LIN {X 0,Y 448.323,Z 386.523,A -85,B 0,C 180,E1 21192.232,E2 21192.232} C_VEL
LIN {X 0,Y 450.072,Z 390.704,A -85,B 0,C 180,E1 21190.556,E2 21190.556} C_VEL
LIN {X 0,Y 452.534,Z 396.687,A -85,B 0,C 180,E1 21188.745,E2 21188.745} C_VEL
LIN {X 0,Y 455.532,Z 405.377,A -85,B 0,C 180,E1 21186.76,E2 21186.76} C_VEL
LIN {X 0,Y 458.055,Z 414.218,A -85,B 0,C 180,E1 21185.151,E2 21185.151} C_VEL
LIN {X 0,Y 453.671,Z 442.774,A -85,B 0,C 180,E1 21182.083,E2 21182.083} C_VEL
LIN {X 0,Y 451.675,Z 461.261,A -85,B 0,C 180,E1 21180.253,E2 21180.253} C_VEL
LIN {X 0,Y 454.574,Z 485.875,A -85,B 0,C 180,E1 21179.545,E2 21179.545} C_VEL
LIN {X 0,Y 450.23,Z 669.654,A -85,B 0,C 180,E1 21176.099,E2 21176.099} C_VEL
LIN {X 0,Y 449.356,Z 688.845,A -85,B 0,C 180,E1 21175.507,E2 21175.507} C_VEL
LIN {X 0,Y 448.327,Z 706.902,A -85,B 0,C 180,E1 21174.719,E2 21174.719} C_VEL
LIN {X 0,Y 447.086,Z 725.176,A -85,B 0,C 180,E1 21173.668,E2 21173.668} C_VEL
LIN {X 0,Y 445.807,Z 742.394,A -85,B 0,C 180,E1 21172.413,E2 21172.413} C_VEL
LIN {X 0,Y 444.541,Z 758.619,A -85,B 0,C 180,E1 21170.954,E2 21170.954} C_VEL
LIN {X 0,Y 443.391,Z 773.227,A -85,B 0,C 180,E1 21169.359,E2 21169.359} C_VEL
LIN {X 0,Y 442.317,Z 787.369,A -85,B 0,C 180,E1 21167.497,E2 21167.497} C_VEL
LIN {X 0,Y 441.437,Z 799.818,A -85,B 0,C 180,E1 21165.502,E2 21165.502} C_VEL
LIN {X 0,Y 440.821,Z 810.693,A -85,B 0,C 180,E1 21163.377,E2 21163.377} C_VEL
LIN {X 0,Y 440.407,Z 819.525,A -85,B 0,C 180,E1 21161.254,E2 21161.254} C_VEL
LIN {X 0,Y 440.196,Z 826.898,A -85,B 0,C 180,E1 21159.017,E2 21159.017} C_VEL
LIN {X 0,Y 440.132,Z 832.486,A -85,B 0,C 180,E1 21156.784,E2 21156.784} C_VEL
LIN {X 0,Y 440.129,Z 836.41,A -85,B 0,C 180,E1 21154.561,E2 21154.561} C_VEL
LIN {X 0,Y 440.162,Z 838.826,A -85,B 0,C 180,E1 21152.213,E2 21152.213} C_VEL
LIN {X 0,Y 440.188,Z 839.52,A -85,B 0,C 180,E1 21149.87,E2 21149.87} C_VEL
LIN {X 0,Y 440.167,Z 838.494,A -85,B 0,C 180,E1 21147.526,E2 21147.526} C_VEL
LIN {X 0,Y 440.145,Z 835.73,A -85,B 0,C 180,E1 21145.179,E2 21145.179} C_VEL
LIN {X 0,Y 440.157,Z 831.15,A -85,B 0,C 180,E1 21142.823,E2 21142.823} C_VEL
LIN {X 0,Y 440.234,Z 825.056,A -85,B 0,C 180,E1 21140.588,E2 21140.588} C_VEL
LIN {X 0,Y 440.458,Z 817.062,A -85,B 0,C 180,E1 21138.344,E2 21138.344} C_VEL
LIN {X 0,Y 440.871,Z 807.59,A -85,B 0,C 180,E1 21136.224,E2 21136.224} C_VEL
LIN {X 0,Y 441.467,Z 796.714,A -85,B 0,C 180,E1 21134.23,E2 21134.23} C_VEL
LIN {X 0,Y 442.299,Z 783.981,A -85,B 0,C 180,E1 21132.299,E2 21132.299} C_VEL
LIN {X 0,Y 443.301,Z 769.666,A -85,B 0,C 180,E1 21130.5,E2 21130.5} C_VEL
LIN {X 0,Y 444.48,Z 753.65,A -85,B 0,C 180,E1 21128.835,E2 21128.835} C_VEL
LIN {X 0,Y 445.682,Z 737.336,A -85,B 0,C 180,E1 21127.441,E2 21127.441} C_VEL
LIN {X 0,Y 446.939,Z 719.499,A -85,B 0,C 180,E1 21126.203,E2 21126.203} C_VEL
LIN {X 0,Y 448.18,Z 700.55,A -85,B 0,C 180,E1 21125.167,E2 21125.167} C_VEL
LIN {X 0,Y 449.289,Z 680.808,A -85,B 0,C 180,E1 21124.364,E2 21124.364} C_VEL
LIN {X 0,Y 450.185,Z 660.789,A -85,B 0,C 180,E1 21123.804,E2 21123.804} C_VEL
LIN {X 0,Y 453.255,Z 560.014,A -85,B 0,C 180,E1 21121.719,E2 21121.719} C_VEL
LIN {X 0,Y 456.39,Z 483.809,A -85,B 0,C 180,E1 21119.981,E2 21119.981} C_VEL
LIN {X 0,Y 453.832,Z 456.502,A -85,B 0,C 180,E1 21118.93,E2 21118.93} C_VEL
LIN {X 0,Y 452.06,Z 438.943,A -85,B 0,C 180,E1 21118.138,E2 21118.138} C_VEL
LIN {X 0,Y 454.372,Z 409.393,A -85,B 0,C 180,E1 21115.386,E2 21115.386} C_VEL
LIN {X 0,Y 446.459,Z 386.782,A -85,B 0,C 180,E1 21112.447,E2 21112.447} C_VEL
LIN {X 0,Y 441.13,Z 371.851,A -85,B 0,C 180,E1 21110.354,E2 21110.354} C_VEL
LIN {X 0,Y 441.125,Z 371.85,A -85,B 0,C 180,E1 21106.624,E2 21106.624} C_VEL
LIN {X 0,Y 441.137,Z 371.849,A -85,B 0,C 180,E1 21102.937,E2 21102.937} C_VEL
LIN {X 0,Y 441.181,Z 371.846,A -85,B 0,C 180,E1 21099.388,E2 21099.388} C_VEL
LIN {X 0,Y 441.156,Z 372.028,A -85,B 0,C 180,E1 21098.847,E2 21098.847} C_VEL
LIN {X 0,Y 442.405,Z 375.286,A -85,B 0,C 180,E1 21098.097,E2 21098.097} C_VEL
LIN {X 0,Y 444.147,Z 377.5,A -85,B 0,C 180,E1 21097.432,E2 21097.432} C_VEL
LIN {X 0,Y 445.923,Z 381.17,A -85,B 0,C 180,E1 21096.609,E2 21096.609} C_VEL
LIN {X 0,Y 448.955,Z 387.643,A -85,B 0,C 180,E1 21095.291,E2 21095.291} C_VEL
LIN {X 0,Y 452.423,Z 396,A -85,B 0,C 180,E1 21093.802,E2 21093.802} C_VEL
LIN {X 0,Y 455.852,Z 406.812,A -85,B 0,C 180,E1 21092.151,E2 21092.151} C_VEL
LIN {X 0,Y 456.831,Z 411.358,A -85,B 0,C 180,E1 21091.54,E2 21091.54} C_VEL
LIN {X 0,Y 456.708,Z 416.112,A -85,B 0,C 180,E1 21091.109,E2 21091.109} C_VEL
LIN {X 0,Y 459.041,Z 430.919,A -85,B 0,C 180,E1 21090.399,E2 21090.399} C_VEL
LIN {X 0,Y 454.36,Z 526.982,A -85,B 0,C 180,E1 21088.206,E2 21088.206} C_VEL
LIN {X 0,Y 451.215,Z 624.113,A -85,B 0,C 180,E1 21086.148,E2 21086.148} C_VEL
LIN {X 0,Y 450.426,Z 643.02,A -85,B 0,C 180,E1 21085.508,E2 21085.508} C_VEL
LIN {X 0,Y 449.445,Z 661.366,A -85,B 0,C 180,E1 21084.653,E2 21084.653} C_VEL
LIN {X 0,Y 448.235,Z 679.768,A -85,B 0,C 180,E1 21083.534,E2 21083.534} C_VEL
LIN {X 0,Y 447.001,Z 696.185,A -85,B 0,C 180,E1 21082.28,E2 21082.28} C_VEL
LIN {X 0,Y 445.732,Z 711.737,A -85,B 0,C 180,E1 21080.827,E2 21080.827} C_VEL
LIN {X 0,Y 444.47,Z 726.31,A -85,B 0,C 180,E1 21079.174,E2 21079.174} C_VEL
LIN {X 0,Y 443.285,Z 739.778,A -85,B 0,C 180,E1 21077.321,E2 21077.321} C_VEL
LIN {X 0,Y 442.267,Z 751.622,A -85,B 0,C 180,E1 21075.338,E2 21075.338} C_VEL
LIN {X 0,Y 441.446,Z 761.933,A -85,B 0,C 180,E1 21073.224,E2 21073.224} C_VEL
LIN {X 0,Y 440.859,Z 770.262,A -85,B 0,C 180,E1 21071.115,E2 21071.115} C_VEL
LIN {X 0,Y 440.452,Z 777.21,A -85,B 0,C 180,E1 21068.88,E2 21068.88} C_VEL
LIN {X 0,Y 440.201,Z 782.678,A -85,B 0,C 180,E1 21066.521,E2 21066.521} C_VEL
LIN {X 0,Y 440.076,Z 786.425,A -85,B 0,C 180,E1 21064.115,E2 21064.115} C_VEL
LIN {X 0,Y 440.031,Z 788.434,A -85,B 0,C 180,E1 21061.693,E2 21061.693} C_VEL
LIN {X 0,Y 440.027,Z 788.727,A -85,B 0,C 180,E1 21059.349,E2 21059.349} C_VEL
LIN {X 0,Y 440.037,Z 787.283,A -85,B 0,C 180,E1 21056.874,E2 21056.874} C_VEL
LIN {X 0,Y 440.1,Z 784.224,A -85,B 0,C 180,E1 21054.524,E2 21054.524} C_VEL
LIN {X 0,Y 440.26,Z 779.442,A -85,B 0,C 180,E1 21052.168,E2 21052.168} C_VEL
LIN {X 0,Y 440.55,Z 773.222,A -85,B 0,C 180,E1 21049.935,E2 21049.935} C_VEL
LIN {X 0,Y 441.035,Z 765.18,A -85,B 0,C 180,E1 21047.695,E2 21047.695} C_VEL
LIN {X 0,Y 441.71,Z 755.698,A -85,B 0,C 180,E1 21045.582,E2 21045.582} C_VEL
LIN {X 0,Y 442.573,Z 744.828,A -85,B 0,C 180,E1 21043.596,E2 21043.596} C_VEL
LIN {X 0,Y 443.616,Z 732.581,A -85,B 0,C 180,E1 21041.742,E2 21041.742} C_VEL
LIN {X 0,Y 444.834,Z 718.548,A -85,B 0,C 180,E1 21039.976,E2 21039.976} C_VEL
LIN {X 0,Y 446.148,Z 703.004,A -85,B 0,C 180,E1 21038.367,E2 21038.367} C_VEL
LIN {X 0,Y 447.44,Z 686.629,A -85,B 0,C 180,E1 21036.979,E2 21036.979} C_VEL
LIN {X 0,Y 448.687,Z 669.284,A -85,B 0,C 180,E1 21035.793,E2 21035.793} C_VEL
LIN {X 0,Y 449.812,Z 650.874,A -85,B 0,C 180,E1 21034.806,E2 21034.806} C_VEL
LIN {X 0,Y 450.73,Z 631.633,A -85,B 0,C 180,E1 21034.038,E2 21034.038} C_VEL
LIN {X 0,Y 451.401,Z 612.37,A -85,B 0,C 180,E1 21033.516,E2 21033.516} C_VEL
LIN {X 0,Y 455.727,Z 428.996,A -85,B 0,C 180,E1 21030.112,E2 21030.112} C_VEL
LIN {X 0,Y 452.048,Z 408.245,A -85,B 0,C 180,E1 21029.421,E2 21029.421} C_VEL
LIN {X 0,Y 452.04,Z 405.292,A -85,B 0,C 180,E1 21029.117,E2 21029.117} C_VEL
LIN {X 0,Y 445.696,Z 385.318,A -85,B 0,C 180,E1 21026.568,E2 21026.568} C_VEL
LIN {X 0,Y 441.168,Z 371.843,A -85,B 0,C 180,E1 21024.774,E2 21024.774} C_VEL
LIN {X 0,Y 441.138,Z 371.849,A -85,B 0,C 180,E1 21021.109,E2 21021.109} C_VEL
LIN {X 0,Y 441.128,Z 371.847,A -85,B 0,C 180,E1 21017.447,E2 21017.447} C_VEL
LIN {X 0,Y 441.133,Z 371.847,A -85,B 0,C 180,E1 21013.694,E2 21013.694} C_VEL
LIN {X 0,Y 441.158,Z 371.846,A -85,B 0,C 180,E1 21010.066,E2 21010.066} C_VEL
LIN {X 0,Y 441.182,Z 371.844,A -85,B 0,C 180,E1 21008.299,E2 21008.299} C_VEL
LIN {X 0,Y 440.154,Z 371.972,A -85,B 0,C 180,E1 21007.299,E2 21007.299} C_VEL
LIN {X 0,Y 433.661,Z 372.783,A -85,B 0,C 180,E1 21004.411,E2 21004.411} C_VEL
LIN {X 0,Y 433.201,Z 372.837,A -85,B 0,C 180,E1 21003.749,E2 21003.749} C_VEL
LIN {X 0,Y 433.227,Z 372.834,A -85,B 0,C 180,E1 21000.055,E2 21000.055} C_VEL
LIN {X 0,Y 433.237,Z 372.832,A -85,B 0,C 180,E1 20996.303,E2 20996.303} C_VEL
LIN {X 0,Y 433.218,Z 372.833,A -85,B 0,C 180,E1 20992.527,E2 20992.527} C_VEL
LIN {X 0,Y 433.195,Z 372.835,A -85,B 0,C 180,E1 20988.853,E2 20988.853} C_VEL
LIN {X 0,Y 433.185,Z 372.836,A -85,B 0,C 180,E1 20985.119,E2 20985.119} C_VEL
LIN {X 0,Y 433.191,Z 372.835,A -85,B 0,C 180,E1 20981.314,E2 20981.314} C_VEL
LIN {X 0,Y 433.215,Z 372.834,A -85,B 0,C 180,E1 20977.693,E2 20977.693} C_VEL
LIN {X 0,Y 433.234,Z 372.83,A -85,B 0,C 180,E1 20973.97,E2 20973.97} C_VEL
LIN {X 0,Y 433.23,Z 372.834,A -85,B 0,C 180,E1 20970.132,E2 20970.132} C_VEL
LIN {X 0,Y 433.201,Z 372.831,A -85,B 0,C 180,E1 20966.427,E2 20966.427} C_VEL
LIN {X 0,Y 433.184,Z 372.831,A -85,B 0,C 180,E1 20962.84,E2 20962.84} C_VEL
LIN {X 0,Y 433.189,Z 372.834,A -85,B 0,C 180,E1 20959.09,E2 20959.09} C_VEL
LIN {X 0,Y 433.212,Z 372.836,A -85,B 0,C 180,E1 20955.429,E2 20955.429} C_VEL
LIN {X 0,Y 433.238,Z 372.836,A -85,B 0,C 180,E1 20951.707,E2 20951.707} C_VEL
LIN {X 0,Y 433.231,Z 372.833,A -85,B 0,C 180,E1 20947.902,E2 20947.902} C_VEL
LIN {X 0,Y 433.204,Z 372.834,A -85,B 0,C 180,E1 20944.137,E2 20944.137} C_VEL
LIN {X 0,Y 433.187,Z 372.834,A -85,B 0,C 180,E1 20940.479,E2 20940.479} C_VEL
LIN {X 0,Y 433.185,Z 372.838,A -85,B 0,C 180,E1 20936.674,E2 20936.674} C_VEL
LIN {X 0,Y 433.196,Z 372.839,A -85,B 0,C 180,E1 20932.957,E2 20932.957} C_VEL
LIN {X 0,Y 433.235,Z 372.836,A -85,B 0,C 180,E1 20929.396,E2 20929.396} C_VEL
LIN {X 0,Y 433.227,Z 372.835,A -85,B 0,C 180,E1 20925.628,E2 20925.628} C_VEL
LIN {X 0,Y 433.21,Z 372.837,A -85,B 0,C 180,E1 20921.838,E2 20921.838} C_VEL
LIN {X 0,Y 433.185,Z 372.838,A -85,B 0,C 180,E1 20918.213,E2 20918.213} C_VEL
LIN {X 0,Y 433.199,Z 372.944,A -85,B 0,C 180,E1 20914.514,E2 20914.514} C_VEL
LIN {X 0,Y 438.764,Z 393.227,A -85,B 0,C 180,E1 20911.037,E2 20911.037} C_VEL
LIN {X 0,Y 441.094,Z 402.817,A -85,B 0,C 180,E1 20909.465,E2 20909.465} C_VEL
LIN {X 0,Y 439.171,Z 430.368,A -85,B 0,C 180,E1 20905.631,E2 20905.631} C_VEL
LIN {X 0,Y 437.342,Z 459.208,A -85,B 0,C 180,E1 20901.672,E2 20901.672} C_VEL
LIN {X 0,Y 436.291,Z 479.402,A -85,B 0,C 180,E1 20898.979,E2 20898.979} C_VEL
LIN {X 0,Y 439.269,Z 500.885,A -85,B 0,C 180,E1 20898.376,E2 20898.376} C_VEL
LIN {X 0,Y 437.139,Z 601.136,A -85,B 0,C 180,E1 20896.315,E2 20896.315} C_VEL
LIN {X 0,Y 436.787,Z 616.364,A -85,B 0,C 180,E1 20895.773,E2 20895.773} C_VEL
LIN {X 0,Y 436.267,Z 632.271,A -85,B 0,C 180,E1 20894.942,E2 20894.942} C_VEL
LIN {X 0,Y 435.587,Z 647.652,A -85,B 0,C 180,E1 20893.839,E2 20893.839} C_VEL
LIN {X 0,Y 434.95,Z 661.323,A -85,B 0,C 180,E1 20892.547,E2 20892.547} C_VEL
LIN {X 0,Y 434.38,Z 672.936,A -85,B 0,C 180,E1 20891.149,E2 20891.149} C_VEL
LIN {X 0,Y 433.908,Z 682.701,A -85,B 0,C 180,E1 20889.684,E2 20889.684} C_VEL
LIN {X 0,Y 433.496,Z 691.731,A -85,B 0,C 180,E1 20887.955,E2 20887.955} C_VEL
LIN {X 0,Y 433.223,Z 698.656,A -85,B 0,C 180,E1 20886.228,E2 20886.228} C_VEL
LIN {X 0,Y 433.06,Z 704.17,A -85,B 0,C 180,E1 20884.37,E2 20884.37} C_VEL
LIN {X 0,Y 432.988,Z 708,A -85,B 0,C 180,E1 20882.382,E2 20882.382} C_VEL
LIN {X 0,Y 433.023,Z 709.862,A -85,B 0,C 180,E1 20880.529,E2 20880.529} C_VEL
LIN {X 0,Y 433.109,Z 710.028,A -85,B 0,C 180,E1 20878.545,E2 20878.545} C_VEL
LIN {X 0,Y 433.284,Z 708.445,A -85,B 0,C 180,E1 20876.693,E2 20876.693} C_VEL
LIN {X 0,Y 433.567,Z 704.888,A -85,B 0,C 180,E1 20874.707,E2 20874.707} C_VEL
LIN {X 0,Y 433.969,Z 699.603,A -85,B 0,C 180,E1 20872.853,E2 20872.853} C_VEL
LIN {X 0,Y 434.461,Z 692.85,A -85,B 0,C 180,E1 20871.13,E2 20871.13} C_VEL
LIN {X 0,Y 435.104,Z 683.912,A -85,B 0,C 180,E1 20869.407,E2 20869.407} C_VEL
LIN {X 0,Y 435.857,Z 673.21,A -85,B 0,C 180,E1 20867.816,E2 20867.816} C_VEL
LIN {X 0,Y 436.602,Z 662.003,A -85,B 0,C 180,E1 20866.492,E2 20866.492} C_VEL
LIN {X 0,Y 437.373,Z 649.291,A -85,B 0,C 180,E1 20865.3,E2 20865.3} C_VEL
LIN {X 0,Y 438.171,Z 634.655,A -85,B 0,C 180,E1 20864.244,E2 20864.244} C_VEL
LIN {X 0,Y 438.804,Z 620.091,A -85,B 0,C 180,E1 20863.452,E2 20863.452} C_VEL
LIN {X 0,Y 439.375,Z 603.875,A -85,B 0,C 180,E1 20862.822,E2 20862.822} C_VEL
LIN {X 0,Y 443.897,Z 510.297,A -85,B 0,C 180,E1 20860.295,E2 20860.295} C_VEL
LIN {X 0,Y 444.177,Z 501.591,A -85,B 0,C 180,E1 20860.039,E2 20860.039} C_VEL
LIN {X 0,Y 440.597,Z 481.46,A -85,B 0,C 180,E1 20859.048,E2 20859.048} C_VEL
LIN {X 0,Y 440.178,Z 478.915,A -85,B 0,C 180,E1 20858.888,E2 20858.888} C_VEL
LIN {X 0,Y 443.155,Z 451.096,A -85,B 0,C 180,E1 20854.759,E2 20854.759} C_VEL
LIN {X 0,Y 446.814,Z 425.609,A -85,B 0,C 180,E1 20850.777,E2 20850.777} C_VEL
LIN {X 0,Y 448.475,Z 415.609,A -85,B 0,C 180,E1 20849.132,E2 20849.132} C_VEL
LIN {X 0,Y 446.478,Z 406.377,A -85,B 0,C 180,E1 20846.878,E2 20846.878} C_VEL
LIN {X 0,Y 444.585,Z 399.623,A -85,B 0,C 180,E1 20844.849,E2 20844.849} C_VEL
LIN {X 0,Y 442.913,Z 394.174,A -85,B 0,C 180,E1 20842.771,E2 20842.771} C_VEL
LIN {X 0,Y 441.579,Z 390.597,A -85,B 0,C 180,E1 20840.822,E2 20840.822} C_VEL
LIN {X 0,Y 440.717,Z 387.966,A -85,B 0,C 180,E1 20838.28,E2 20838.28} C_VEL
LIN {X 0,Y 440.834,Z 387.574,A -85,B 0,C 180,E1 20836.347,E2 20836.347} C_VEL
LIN {X 0,Y 441.244,Z 389.399,A -85,B 0,C 180,E1 20834.261,E2 20834.261} C_VEL
LIN {X 0,Y 442.742,Z 392.108,A -85,B 0,C 180,E1 20832.398,E2 20832.398} C_VEL
LIN {X 0,Y 444.376,Z 396.253,A -85,B 0,C 180,E1 20830.689,E2 20830.689} C_VEL
LIN {X 0,Y 446.617,Z 401.89,A -85,B 0,C 180,E1 20828.926,E2 20828.926} C_VEL
LIN {X 0,Y 449.341,Z 410.137,A -85,B 0,C 180,E1 20826.981,E2 20826.981} C_VEL
LIN {X 0,Y 451.373,Z 417.564,A -85,B 0,C 180,E1 20825.555,E2 20825.555} C_VEL
LIN {X 0,Y 446.824,Z 444.559,A -85,B 0,C 180,E1 20822.559,E2 20822.559} C_VEL
LIN {X 0,Y 444.658,Z 462.787,A -85,B 0,C 180,E1 20820.706,E2 20820.706} C_VEL
LIN {X 0,Y 447.451,Z 486.897,A -85,B 0,C 180,E1 20819.997,E2 20819.997} C_VEL
LIN {X 0,Y 442.821,Z 669.243,A -85,B 0,C 180,E1 20816.493,E2 20816.493} C_VEL
LIN {X 0,Y 441.899,Z 688.487,A -85,B 0,C 180,E1 20815.889,E2 20815.889} C_VEL
LIN {X 0,Y 440.738,Z 707.541,A -85,B 0,C 180,E1 20815.036,E2 20815.036} C_VEL
LIN {X 0,Y 439.435,Z 725.675,A -85,B 0,C 180,E1 20813.963,E2 20813.963} C_VEL
LIN {X 0,Y 438.094,Z 742.722,A -85,B 0,C 180,E1 20812.688,E2 20812.688} C_VEL
LIN {X 0,Y 436.764,Z 758.821,A -85,B 0,C 180,E1 20811.205,E2 20811.205} C_VEL
LIN {X 0,Y 435.508,Z 773.914,A -85,B 0,C 180,E1 20809.515,E2 20809.515} C_VEL
LIN {X 0,Y 434.408,Z 787.594,A -85,B 0,C 180,E1 20807.658,E2 20807.658} C_VEL
LIN {X 0,Y 433.497,Z 799.794,A -85,B 0,C 180,E1 20805.656,E2 20805.656} C_VEL
LIN {X 0,Y 432.848,Z 810.623,A -85,B 0,C 180,E1 20803.492,E2 20803.492} C_VEL
LIN {X 0,Y 432.417,Z 819.378,A -85,B 0,C 180,E1 20801.335,E2 20801.335} C_VEL
LIN {X 0,Y 432.2,Z 826.71,A -85,B 0,C 180,E1 20799.051,E2 20799.051} C_VEL
LIN {X 0,Y 432.136,Z 832.237,A -85,B 0,C 180,E1 20796.777,E2 20796.777} C_VEL
LIN {X 0,Y 432.137,Z 836.092,A -85,B 0,C 180,E1 20794.512,E2 20794.512} C_VEL
LIN {X 0,Y 432.177,Z 838.428,A -85,B 0,C 180,E1 20792.121,E2 20792.121} C_VEL
LIN {X 0,Y 432.201,Z 839.059,A -85,B 0,C 180,E1 20789.867,E2 20789.867} C_VEL
LIN {X 0,Y 432.178,Z 838.023,A -85,B 0,C 180,E1 20787.481,E2 20787.481} C_VEL
LIN {X 0,Y 432.153,Z 835.238,A -85,B 0,C 180,E1 20785.089,E2 20785.089} C_VEL
LIN {X 0,Y 432.162,Z 830.63,A -85,B 0,C 180,E1 20782.689,E2 20782.689} C_VEL
LIN {X 0,Y 432.242,Z 824.498,A -85,B 0,C 180,E1 20780.413,E2 20780.413} C_VEL
LIN {X 0,Y 432.492,Z 816.466,A -85,B 0,C 180,E1 20778.126,E2 20778.126} C_VEL
LIN {X 0,Y 432.953,Z 806.704,A -85,B 0,C 180,E1 20775.917,E2 20775.917} C_VEL
LIN {X 0,Y 433.643,Z 795.207,A -85,B 0,C 180,E1 20773.8,E2 20773.8} C_VEL
LIN {X 0,Y 434.542,Z 782.451,A -85,B 0,C 180,E1 20771.858,E2 20771.858} C_VEL
LIN {X 0,Y 435.709,Z 767.172,A -85,B 0,C 180,E1 20769.938,E2 20769.938} C_VEL
LIN {X 0,Y 436.965,Z 751.461,A -85,B 0,C 180,E1 20768.312,E2 20768.312} C_VEL
LIN {X 0,Y 438.285,Z 734.851,A -85,B 0,C 180,E1 20766.897,E2 20766.897} C_VEL
LIN {X 0,Y 439.618,Z 717.425,A -85,B 0,C 180,E1 20765.691,E2 20765.691} C_VEL
LIN {X 0,Y 440.946,Z 698.444,A -85,B 0,C 180,E1 20764.659,E2 20764.659} C_VEL
LIN {X 0,Y 442.114,Z 679.134,A -85,B 0,C 180,E1 20763.872,E2 20763.872} C_VEL
LIN {X 0,Y 443.11,Z 658.21,A -85,B 0,C 180,E1 20763.286,E2 20763.286} C_VEL
LIN {X 0,Y 446.286,Z 564.966,A -85,B 0,C 180,E1 20761.282,E2 20761.282} C_VEL
LIN {X 0,Y 449.994,Z 485.057,A -85,B 0,C 180,E1 20759.39,E2 20759.39} C_VEL
LIN {X 0,Y 447.773,Z 458.476,A -85,B 0,C 180,E1 20758.315,E2 20758.315} C_VEL
LIN {X 0,Y 445.642,Z 436.943,A -85,B 0,C 180,E1 20757.284,E2 20757.284} C_VEL
LIN {X 0,Y 445.354,Z 431.936,A -85,B 0,C 180,E1 20757.014,E2 20757.014} C_VEL
LIN {X 0,Y 447.108,Z 412.354,A -85,B 0,C 180,E1 20755.156,E2 20755.156} C_VEL
LIN {X 0,Y 439.234,Z 389.836,A -85,B 0,C 180,E1 20752.176,E2 20752.176} C_VEL
LIN {X 0,Y 433.234,Z 372.834,A -85,B 0,C 180,E1 20749.743,E2 20749.743} C_VEL
LIN {X 0,Y 433.207,Z 372.837,A -85,B 0,C 180,E1 20745.995,E2 20745.995} C_VEL
LIN {X 0,Y 433.186,Z 372.84,A -85,B 0,C 180,E1 20742.375,E2 20742.375} C_VEL
LIN {X 0,Y 433.229,Z 372.96,A -85,B 0,C 180,E1 20741.129,E2 20741.129} C_VEL
LIN {X 0,Y 434.369,Z 376.125,A -85,B 0,C 180,E1 20740.13,E2 20740.13} C_VEL
LIN {X 0,Y 436.626,Z 378.792,A -85,B 0,C 180,E1 20739.031,E2 20739.031} C_VEL
LIN {X 0,Y 438.281,Z 382.311,A -85,B 0,C 180,E1 20738.088,E2 20738.088} C_VEL
LIN {X 0,Y 439.316,Z 383.882,A -85,B 0,C 180,E1 20737.624,E2 20737.624} C_VEL
LIN {X 0,Y 442.999,Z 391.548,A -85,B 0,C 180,E1 20735.877,E2 20735.877} C_VEL
LIN {X 0,Y 446.758,Z 401.149,A -85,B 0,C 180,E1 20734.098,E2 20734.098} C_VEL
LIN {X 0,Y 450.019,Z 412.107,A -85,B 0,C 180,E1 20732.375,E2 20732.375} C_VEL
LIN {X 0,Y 450.516,Z 415.208,A -85,B 0,C 180,E1 20731.959,E2 20731.959} C_VEL
LIN {X 0,Y 450.676,Z 417.731,A -85,B 0,C 180,E1 20731.77,E2 20731.77} C_VEL
LIN {X 0,Y 452.867,Z 432.571,A -85,B 0,C 180,E1 20731.019,E2 20731.019} C_VEL
LIN {X 0,Y 447.682,Z 527.539,A -85,B 0,C 180,E1 20728.761,E2 20728.761} C_VEL
LIN {X 0,Y 444.512,Z 612.909,A -85,B 0,C 180,E1 20726.907,E2 20726.907} C_VEL
LIN {X 0,Y 443.77,Z 633.282,A -85,B 0,C 180,E1 20726.35,E2 20726.35} C_VEL
LIN {X 0,Y 442.811,Z 652.164,A -85,B 0,C 180,E1 20725.584,E2 20725.584} C_VEL
LIN {X 0,Y 441.665,Z 670.105,A -85,B 0,C 180,E1 20724.617,E2 20724.617} C_VEL
LIN {X 0,Y 440.339,Z 687.622,A -85,B 0,C 180,E1 20723.413,E2 20723.413} C_VEL
LIN {X 0,Y 438.965,Z 703.963,A -85,B 0,C 180,E1 20722.02,E2 20722.02} C_VEL
LIN {X 0,Y 437.608,Z 718.963,A -85,B 0,C 180,E1 20720.461,E2 20720.461} C_VEL
LIN {X 0,Y 436.3,Z 732.873,A -85,B 0,C 180,E1 20718.713,E2 20718.713} C_VEL
LIN {X 0,Y 435.133,Z 745.286,A -85,B 0,C 180,E1 20716.829,E2 20716.829} C_VEL
LIN {X 0,Y 434.139,Z 756.275,A -85,B 0,C 180,E1 20714.812,E2 20714.812} C_VEL
LIN {X 0,Y 433.307,Z 766.218,A -85,B 0,C 180,E1 20712.557,E2 20712.557} C_VEL
LIN {X 0,Y 432.732,Z 774.275,A -85,B 0,C 180,E1 20710.248,E2 20710.248} C_VEL
LIN {X 0,Y 432.38,Z 780.39,A -85,B 0,C 180,E1 20707.975,E2 20707.975} C_VEL
LIN {X 0,Y 432.17,Z 785.041,A -85,B 0,C 180,E1 20705.576,E2 20705.576} C_VEL
LIN {X 0,Y 432.073,Z 787.96,A -85,B 0,C 180,E1 20703.184,E2 20703.184} C_VEL
LIN {X 0,Y 432.041,Z 789.227,A -85,B 0,C 180,E1 20700.795,E2 20700.795} C_VEL
LIN {X 0,Y 432.032,Z 788.863,A -85,B 0,C 180,E1 20698.408,E2 20698.408} C_VEL
LIN {X 0,Y 432.063,Z 786.867,A -85,B 0,C 180,E1 20696.019,E2 20696.019} C_VEL
LIN {X 0,Y 432.165,Z 783.193,A -85,B 0,C 180,E1 20693.624,E2 20693.624} C_VEL
LIN {X 0,Y 432.388,Z 777.743,A -85,B 0,C 180,E1 20691.221,E2 20691.221} C_VEL
LIN {X 0,Y 432.798,Z 770.367,A -85,B 0,C 180,E1 20688.81,E2 20688.81} C_VEL
LIN {X 0,Y 433.42,Z 761.407,A -85,B 0,C 180,E1 20686.526,E2 20686.526} C_VEL
LIN {X 0,Y 434.262,Z 750.917,A -85,B 0,C 180,E1 20684.372,E2 20684.372} C_VEL
LIN {X 0,Y 435.316,Z 738.919,A -85,B 0,C 180,E1 20682.351,E2 20682.351} C_VEL
LIN {X 0,Y 436.549,Z 725.351,A -85,B 0,C 180,E1 20680.464,E2 20680.464} C_VEL
LIN {X 0,Y 437.867,Z 710.663,A -85,B 0,C 180,E1 20678.781,E2 20678.781} C_VEL
LIN {X 0,Y 439.202,Z 695.033,A -85,B 0,C 180,E1 20677.302,E2 20677.302} C_VEL
LIN {X 0,Y 440.509,Z 678.572,A -85,B 0,C 180,E1 20676.028,E2 20676.028} C_VEL
LIN {X 0,Y 441.725,Z 661.354,A -85,B 0,C 180,E1 20674.958,E2 20674.958} C_VEL
LIN {X 0,Y 442.816,Z 642.343,A -85,B 0,C 180,E1 20674.048,E2 20674.048} C_VEL
LIN {X 0,Y 443.672,Z 622.983,A -85,B 0,C 180,E1 20673.381,E2 20673.381} C_VEL
LIN {X 0,Y 444.284,Z 600.977,A -85,B 0,C 180,E1 20672.9,E2 20672.9} C_VEL
LIN {X 0,Y 448.679,Z 430.475,A -85,B 0,C 180,E1 20669.664,E2 20669.664} C_VEL
LIN {X 0,Y 444.852,Z 408.471,A -85,B 0,C 180,E1 20668.909,E2 20668.909} C_VEL
LIN {X 0,Y 438.598,Z 388.705,A -85,B 0,C 180,E1 20666.361,E2 20666.361} C_VEL
LIN {X 0,Y 433.219,Z 372.832,A -85,B 0,C 180,E1 20664.232,E2 20664.232} C_VEL
LIN {X 0,Y 433.246,Z 372.828,A -85,B 0,C 180,E1 20660.428,E2 20660.428} C_VEL
LIN {X 0,Y 433.238,Z 372.835,A -85,B 0,C 180,E1 20656.548,E2 20656.548} C_VEL
LIN {X 0,Y 433.221,Z 372.834,A -85,B 0,C 180,E1 20652.73,E2 20652.73} C_VEL
LIN {X 0,Y 433.192,Z 372.835,A -85,B 0,C 180,E1 20649.147,E2 20649.147} C_VEL
LIN {X 0,Y 433.189,Z 372.836,A -85,B 0,C 180,E1 20645.405,E2 20645.405} C_VEL
LIN {X 0,Y 433.201,Z 372.837,A -85,B 0,C 180,E1 20643.749,E2 20643.749} C_VEL
LIN {X 0,Y 432.174,Z 372.966,A -85,B 0,C 180,E1 20642.73,E2 20642.73} C_VEL
LIN {X 0,Y 425.675,Z 373.774,A -85,B 0,C 180,E1 20639.786,E2 20639.786} C_VEL
LIN {X 0,Y 425.251,Z 373.822,A -85,B 0,C 180,E1 20639.111,E2 20639.111} C_VEL
LIN {X 0,Y 425.251,Z 373.824,A -85,B 0,C 180,E1 20635.336,E2 20635.336} C_VEL
LIN {X 0,Y 425.265,Z 373.822,A -85,B 0,C 180,E1 20631.662,E2 20631.662} C_VEL
LIN {X 0,Y 425.288,Z 373.821,A -85,B 0,C 180,E1 20627.938,E2 20627.938} C_VEL
LIN {X 0,Y 425.307,Z 373.822,A -85,B 0,C 180,E1 20624.152,E2 20624.152} C_VEL
LIN {X 0,Y 425.286,Z 373.824,A -85,B 0,C 180,E1 20620.293,E2 20620.293} C_VEL
LIN {X 0,Y 425.261,Z 373.822,A -85,B 0,C 180,E1 20616.616,E2 20616.616} C_VEL
LIN {X 0,Y 425.248,Z 373.82,A -85,B 0,C 180,E1 20612.83,E2 20612.83} C_VEL
LIN {X 0,Y 425.247,Z 373.82,A -85,B 0,C 180,E1 20609.057,E2 20609.057} C_VEL
LIN {X 0,Y 425.255,Z 373.823,A -85,B 0,C 180,E1 20605.28,E2 20605.28} C_VEL
LIN {X 0,Y 425.283,Z 373.823,A -85,B 0,C 180,E1 20601.618,E2 20601.618} C_VEL
LIN {X 0,Y 425.295,Z 373.821,A -85,B 0,C 180,E1 20597.784,E2 20597.784} C_VEL
LIN {X 0,Y 425.283,Z 373.825,A -85,B 0,C 180,E1 20594.034,E2 20594.034} C_VEL
LIN {X 0,Y 425.257,Z 373.825,A -85,B 0,C 180,E1 20590.353,E2 20590.353} C_VEL
LIN {X 0,Y 425.248,Z 373.823,A -85,B 0,C 180,E1 20586.733,E2 20586.733} C_VEL
LIN {X 0,Y 425.249,Z 373.823,A -85,B 0,C 180,E1 20582.862,E2 20582.862} C_VEL
LIN {X 0,Y 425.265,Z 373.826,A -85,B 0,C 180,E1 20579.166,E2 20579.166} C_VEL
LIN {X 0,Y 425.284,Z 373.828,A -85,B 0,C 180,E1 20575.373,E2 20575.373} C_VEL
LIN {X 0,Y 425.302,Z 373.825,A -85,B 0,C 180,E1 20571.464,E2 20571.464} C_VEL
LIN {X 0,Y 425.296,Z 373.824,A -85,B 0,C 180,E1 20567.567,E2 20567.567} C_VEL
LIN {X 0,Y 425.28,Z 373.824,A -85,B 0,C 180,E1 20563.726,E2 20563.726} C_VEL
LIN {X 0,Y 425.253,Z 373.827,A -85,B 0,C 180,E1 20560.108,E2 20560.108} C_VEL
LIN {X 0,Y 425.245,Z 373.828,A -85,B 0,C 180,E1 20556.336,E2 20556.336} C_VEL
LIN {X 0,Y 425.288,Z 373.946,A -85,B 0,C 180,E1 20555.005,E2 20555.005} C_VEL
LIN {X 0,Y 430.687,Z 393.583,A -85,B 0,C 180,E1 20551.569,E2 20551.569} C_VEL
LIN {X 0,Y 433.505,Z 405.126,A -85,B 0,C 180,E1 20549.652,E2 20549.652} C_VEL
LIN {X 0,Y 431.51,Z 432.213,A -85,B 0,C 180,E1 20545.825,E2 20545.825} C_VEL
LIN {X 0,Y 429.612,Z 460.708,A -85,B 0,C 180,E1 20541.863,E2 20541.863} C_VEL
LIN {X 0,Y 428.589,Z 479.295,A -85,B 0,C 180,E1 20539.349,E2 20539.349} C_VEL
LIN {X 0,Y 431.665,Z 501.721,A -85,B 0,C 180,E1 20538.696,E2 20538.696} C_VEL
LIN {X 0,Y 429.405,Z 601.912,A -85,B 0,C 180,E1 20536.573,E2 20536.573} C_VEL
LIN {X 0,Y 429.026,Z 617.345,A -85,B 0,C 180,E1 20536.007,E2 20536.007} C_VEL
LIN {X 0,Y 428.475,Z 633.333,A -85,B 0,C 180,E1 20535.151,E2 20535.151} C_VEL
LIN {X 0,Y 427.793,Z 648.182,A -85,B 0,C 180,E1 20534.068,E2 20534.068} C_VEL
LIN {X 0,Y 427.136,Z 661.7,A -85,B 0,C 180,E1 20532.78,E2 20532.78} C_VEL
LIN {X 0,Y 426.595,Z 672.485,A -85,B 0,C 180,E1 20531.492,E2 20531.492} C_VEL
LIN {X 0,Y 426.041,Z 683.372,A -85,B 0,C 180,E1 20529.865,E2 20529.865} C_VEL
LIN {X 0,Y 425.606,Z 692.527,A -85,B 0,C 180,E1 20528.103,E2 20528.103} C_VEL
LIN {X 0,Y 425.317,Z 699.567,A -85,B 0,C 180,E1 20526.344,E2 20526.344} C_VEL
LIN {X 0,Y 425.146,Z 705.183,A -85,B 0,C 180,E1 20524.451,E2 20524.451} C_VEL
LIN {X 0,Y 425.072,Z 709.114,A -85,B 0,C 180,E1 20522.427,E2 20522.427} C_VEL
LIN {X 0,Y 425.114,Z 711.059,A -85,B 0,C 180,E1 20520.539,E2 20520.539} C_VEL
LIN {X 0,Y 425.213,Z 711.295,A -85,B 0,C 180,E1 20518.518,E2 20518.518} C_VEL
LIN {X 0,Y 425.413,Z 709.802,A -85,B 0,C 180,E1 20516.632,E2 20516.632} C_VEL
LIN {X 0,Y 425.728,Z 706.313,A -85,B 0,C 180,E1 20514.61,E2 20514.61} C_VEL
LIN {X 0,Y 426.169,Z 701.084,A -85,B 0,C 180,E1 20512.722,E2 20512.722} C_VEL
LIN {X 0,Y 426.708,Z 694.398,A -85,B 0,C 180,E1 20510.968,E2 20510.968} C_VEL
LIN {X 0,Y 427.411,Z 685.574,A -85,B 0,C 180,E1 20509.214,E2 20509.214} C_VEL
LIN {X 0,Y 428.158,Z 676.024,A -85,B 0,C 180,E1 20507.731,E2 20507.731} C_VEL
LIN {X 0,Y 429.033,Z 663.977,A -85,B 0,C 180,E1 20506.249,E2 20506.249} C_VEL
LIN {X 0,Y 429.953,Z 649.904,A -85,B 0,C 180,E1 20504.903,E2 20504.903} C_VEL
LIN {X 0,Y 430.886,Z 634.249,A -85,B 0,C 180,E1 20503.763,E2 20503.763} C_VEL
LIN {X 0,Y 431.649,Z 617.938,A -85,B 0,C 180,E1 20502.892,E2 20502.892} C_VEL
LIN {X 0,Y 432.264,Z 600.365,A -85,B 0,C 180,E1 20502.257,E2 20502.257} C_VEL
LIN {X 0,Y 437.302,Z 508.055,A -85,B 0,C 180,E1 20499.668,E2 20499.668} C_VEL
LIN {X 0,Y 437.375,Z 502.766,A -85,B 0,C 180,E1 20499.492,E2 20499.492} C_VEL
LIN {X 0,Y 433.792,Z 482.149,A -85,B 0,C 180,E1 20498.419,E2 20498.419} C_VEL
LIN {X 0,Y 433.197,Z 478.683,A -85,B 0,C 180,E1 20498.186,E2 20498.186} C_VEL
LIN {X 0,Y 436.325,Z 452.451,A -85,B 0,C 180,E1 20494.19,E2 20494.19} C_VEL
LIN {X 0,Y 440.321,Z 427.366,A -85,B 0,C 180,E1 20490.162,E2 20490.162} C_VEL
LIN {X 0,Y 441.8,Z 419.252,A -85,B 0,C 180,E1 20488.784,E2 20488.784} C_VEL
LIN {X 0,Y 439.964,Z 410.313,A -85,B 0,C 180,E1 20486.479,E2 20486.479} C_VEL
LIN {X 0,Y 438.252,Z 403.947,A -85,B 0,C 180,E1 20484.425,E2 20484.425} C_VEL
LIN {X 0,Y 436.75,Z 398.946,A -85,B 0,C 180,E1 20482.32,E2 20482.32} C_VEL
LIN {X 0,Y 435.838,Z 396.085,A -85,B 0,C 180,E1 20480.635,E2 20480.635} C_VEL
LIN {X 0,Y 435.226,Z 393.597,A -85,B 0,C 180,E1 20477.87,E2 20477.87} C_VEL
LIN {X 0,Y 435.414,Z 393.609,A -85,B 0,C 180,E1 20476.093,E2 20476.093} C_VEL
LIN {X 0,Y 436.044,Z 395.893,A -85,B 0,C 180,E1 20473.828,E2 20473.828} C_VEL
LIN {X 0,Y 437.213,Z 398.026,A -85,B 0,C 180,E1 20472.426,E2 20472.426} C_VEL
LIN {X 0,Y 438.813,Z 402.262,A -85,B 0,C 180,E1 20470.668,E2 20470.668} C_VEL
LIN {X 0,Y 440.788,Z 407.444,A -85,B 0,C 180,E1 20469.022,E2 20469.022} C_VEL
LIN {X 0,Y 443.144,Z 414.887,A -85,B 0,C 180,E1 20467.206,E2 20467.206} C_VEL
LIN {X 0,Y 444.754,Z 421.402,A -85,B 0,C 180,E1 20465.928,E2 20465.928} C_VEL
LIN {X 0,Y 439.87,Z 447.895,A -85,B 0,C 180,E1 20462.906,E2 20462.906} C_VEL
LIN {X 0,Y 437.679,Z 464.561,A -85,B 0,C 180,E1 20461.159,E2 20461.159} C_VEL
LIN {X 0,Y 440.336,Z 487.827,A -85,B 0,C 180,E1 20460.46,E2 20460.46} C_VEL
LIN {X 0,Y 435.401,Z 669.084,A -85,B 0,C 180,E1 20456.886,E2 20456.886} C_VEL
LIN {X 0,Y 434.417,Z 688.45,A -85,B 0,C 180,E1 20456.263,E2 20456.263} C_VEL
LIN {X 0,Y 433.231,Z 706.909,A -85,B 0,C 180,E1 20455.422,E2 20455.422} C_VEL
LIN {X 0,Y 431.863,Z 724.993,A -85,B 0,C 180,E1 20454.338,E2 20454.338} C_VEL
LIN {X 0,Y 430.455,Z 742.104,A -85,B 0,C 180,E1 20453.041,E2 20453.041} C_VEL
LIN {X 0,Y 429.05,Z 758.263,A -85,B 0,C 180,E1 20451.533,E2 20451.533} C_VEL
LIN {X 0,Y 427.723,Z 773.411,A -85,B 0,C 180,E1 20449.813,E2 20449.813} C_VEL
LIN {X 0,Y 426.528,Z 787.456,A -85,B 0,C 180,E1 20447.873,E2 20447.873} C_VEL
LIN {X 0,Y 425.559,Z 799.73,A -85,B 0,C 180,E1 20445.816,E2 20445.816} C_VEL
LIN {X 0,Y 424.909,Z 809.908,A -85,B 0,C 180,E1 20443.749,E2 20443.749} C_VEL
LIN {X 0,Y 424.438,Z 818.971,A -85,B 0,C 180,E1 20441.484,E2 20441.484} C_VEL
LIN {X 0,Y 424.214,Z 826.134,A -85,B 0,C 180,E1 20439.223,E2 20439.223} C_VEL
LIN {X 0,Y 424.146,Z 831.709,A -85,B 0,C 180,E1 20436.905,E2 20436.905} C_VEL
LIN {X 0,Y 424.146,Z 835.599,A -85,B 0,C 180,E1 20434.597,E2 20434.597} C_VEL
LIN {X 0,Y 424.188,Z 837.956,A -85,B 0,C 180,E1 20432.161,E2 20432.161} C_VEL
LIN {X 0,Y 424.215,Z 838.596,A -85,B 0,C 180,E1 20429.865,E2 20429.865} C_VEL
LIN {X 0,Y 424.188,Z 837.557,A -85,B 0,C 180,E1 20427.433,E2 20427.433} C_VEL
LIN {X 0,Y 424.16,Z 834.757,A -85,B 0,C 180,E1 20424.996,E2 20424.996} C_VEL
LIN {X 0,Y 424.163,Z 830.126,A -85,B 0,C 180,E1 20422.551,E2 20422.551} C_VEL
LIN {X 0,Y 424.253,Z 823.966,A -85,B 0,C 180,E1 20420.23,E2 20420.23} C_VEL
LIN {X 0,Y 424.533,Z 815.903,A -85,B 0,C 180,E1 20417.9,E2 20417.9} C_VEL
LIN {X 0,Y 425.017,Z 806.355,A -85,B 0,C 180,E1 20415.699,E2 20415.699} C_VEL
LIN {X 0,Y 425.728,Z 795.404,A -85,B 0,C 180,E1 20413.63,E2 20413.63} C_VEL
LIN {X 0,Y 426.699,Z 782.575,A -85,B 0,C 180,E1 20411.625,E2 20411.625} C_VEL
LIN {X 0,Y 427.876,Z 768.246,A -85,B 0,C 180,E1 20409.766,E2 20409.766} C_VEL
LIN {X 0,Y 429.257,Z 752.205,A -85,B 0,C 180,E1 20408.047,E2 20408.047} C_VEL
LIN {X 0,Y 430.656,Z 735.897,A -85,B 0,C 180,E1 20406.608,E2 20406.608} C_VEL
LIN {X 0,Y 432.066,Z 718.918,A -85,B 0,C 180,E1 20405.383,E2 20405.383} C_VEL
LIN {X 0,Y 433.524,Z 700.122,A -85,B 0,C 180,E1 20404.304,E2 20404.304} C_VEL
LIN {X 0,Y 434.85,Z 680.523,A -85,B 0,C 180,E1 20403.455,E2 20403.455} C_VEL
LIN {X 0,Y 435.958,Z 660.25,A -85,B 0,C 180,E1 20402.845,E2 20402.845} C_VEL
LIN {X 0,Y 439.515,Z 567.609,A -85,B 0,C 180,E1 20400.765,E2 20400.765} C_VEL
LIN {X 0,Y 443.753,Z 486.38,A -85,B 0,C 180,E1 20398.768,E2 20398.768} C_VEL
LIN {X 0,Y 441.651,Z 458.161,A -85,B 0,C 180,E1 20397.572,E2 20397.572} C_VEL
LIN {X 0,Y 439.811,Z 437.002,A -85,B 0,C 180,E1 20396.498,E2 20396.498} C_VEL
LIN {X 0,Y 439.016,Z 422.457,A -85,B 0,C 180,E1 20395.61,E2 20395.61} C_VEL
LIN {X 0,Y 439.693,Z 414.911,A -85,B 0,C 180,E1 20394.878,E2 20394.878} C_VEL
LIN {X 0,Y 431.434,Z 391.19,A -85,B 0,C 180,E1 20391.673,E2 20391.673} C_VEL
LIN {X 0,Y 430.047,Z 387.1,A -85,B 0,C 180,E1 20391.052,E2 20391.052} C_VEL
LIN {X 0,Y 428.697,Z 379.426,A -85,B 0,C 180,E1 20389.404,E2 20389.404} C_VEL
LIN {X 0,Y 426.437,Z 377.085,A -85,B 0,C 180,E1 20387.213,E2 20387.213} C_VEL
LIN {X 0,Y 426.072,Z 376.423,A -85,B 0,C 180,E1 20385.32,E2 20385.32} C_VEL
LIN {X 0,Y 426.931,Z 377.78,A -85,B 0,C 180,E1 20383.251,E2 20383.251} C_VEL
LIN {X 0,Y 429.269,Z 379.975,A -85,B 0,C 180,E1 20381.307,E2 20381.307} C_VEL
LIN {X 0,Y 430.517,Z 383.213,A -85,B 0,C 180,E1 20380.173,E2 20380.173} C_VEL
LIN {X 0,Y 432.105,Z 384.96,A -85,B 0,C 180,E1 20379.347,E2 20379.347} C_VEL
LIN {X 0,Y 433.656,Z 388.598,A -85,B 0,C 180,E1 20378.332,E2 20378.332} C_VEL
LIN {X 0,Y 434.665,Z 390.424,A -85,B 0,C 180,E1 20377.8,E2 20377.8} C_VEL
LIN {X 0,Y 437.838,Z 397.246,A -85,B 0,C 180,E1 20376.17,E2 20376.17} C_VEL
LIN {X 0,Y 441.3,Z 406.738,A -85,B 0,C 180,E1 20374.344,E2 20374.344} C_VEL
LIN {X 0,Y 444.293,Z 417.486,A -85,B 0,C 180,E1 20372.623,E2 20372.623} C_VEL
LIN {X 0,Y 445.226,Z 421.594,A -85,B 0,C 180,E1 20372.343,E2 20372.343} C_VEL
LIN {X 0,Y 446.873,Z 434.391,A -85,B 0,C 180,E1 20371.67,E2 20371.67} C_VEL
LIN {X 0,Y 441.253,Z 525.936,A -85,B 0,C 180,E1 20369.402,E2 20369.402} C_VEL
LIN {X 0,Y 437.76,Z 607.042,A -85,B 0,C 180,E1 20367.554,E2 20367.554} C_VEL
LIN {X 0,Y 436.925,Z 629.5,A -85,B 0,C 180,E1 20366.98,E2 20366.98} C_VEL
LIN {X 0,Y 435.936,Z 648.753,A -85,B 0,C 180,E1 20366.241,E2 20366.241} C_VEL
LIN {X 0,Y 434.688,Z 667.65,A -85,B 0,C 180,E1 20365.257,E2 20365.257} C_VEL
LIN {X 0,Y 433.334,Z 684.845,A -85,B 0,C 180,E1 20364.104,E2 20364.104} C_VEL
LIN {X 0,Y 431.883,Z 701.17,A -85,B 0,C 180,E1 20362.744,E2 20362.744} C_VEL
LIN {X 0,Y 430.393,Z 716.571,A -85,B 0,C 180,E1 20361.177,E2 20361.177} C_VEL
LIN {X 0,Y 428.937,Z 730.944,A -85,B 0,C 180,E1 20359.4,E2 20359.4} C_VEL
LIN {X 0,Y 427.589,Z 744.18,A -85,B 0,C 180,E1 20357.416,E2 20357.416} C_VEL
LIN {X 0,Y 426.481,Z 755.446,A -85,B 0,C 180,E1 20355.362,E2 20355.362} C_VEL
LIN {X 0,Y 425.589,Z 765.255,A -85,B 0,C 180,E1 20353.173,E2 20353.173} C_VEL
LIN {X 0,Y 424.923,Z 773.573,A -85,B 0,C 180,E1 20350.85,E2 20350.85} C_VEL
LIN {X 0,Y 424.474,Z 780.374,A -85,B 0,C 180,E1 20348.379,E2 20348.379} C_VEL
LIN {X 0,Y 424.224,Z 785.178,A -85,B 0,C 180,E1 20345.945,E2 20345.945} C_VEL
LIN {X 0,Y 424.105,Z 788.254,A -85,B 0,C 180,E1 20343.514,E2 20343.514} C_VEL
LIN {X 0,Y 424.057,Z 789.677,A -85,B 0,C 180,E1 20341.081,E2 20341.081} C_VEL
LIN {X 0,Y 424.045,Z 789.46,A -85,B 0,C 180,E1 20338.649,E2 20338.649} C_VEL
LIN {X 0,Y 424.073,Z 787.603,A -85,B 0,C 180,E1 20336.215,E2 20336.215} C_VEL
LIN {X 0,Y 424.174,Z 784.064,A -85,B 0,C 180,E1 20333.775,E2 20333.775} C_VEL
LIN {X 0,Y 424.398,Z 778.746,A -85,B 0,C 180,E1 20331.328,E2 20331.328} C_VEL
LIN {X 0,Y 424.799,Z 771.816,A -85,B 0,C 180,E1 20328.964,E2 20328.964} C_VEL
LIN {X 0,Y 425.414,Z 763.19,A -85,B 0,C 180,E1 20326.665,E2 20326.665} C_VEL
LIN {X 0,Y 426.252,Z 753.054,A -85,B 0,C 180,E1 20324.49,E2 20324.49} C_VEL
LIN {X 0,Y 427.311,Z 741.365,A -85,B 0,C 180,E1 20322.431,E2 20322.431} C_VEL
LIN {X 0,Y 428.59,Z 727.907,A -85,B 0,C 180,E1 20320.475,E2 20320.475} C_VEL
LIN {X 0,Y 429.969,Z 713.383,A -85,B 0,C 180,E1 20318.73,E2 20318.73} C_VEL
LIN {X 0,Y 431.417,Z 697.526,A -85,B 0,C 180,E1 20317.157,E2 20317.157} C_VEL
LIN {X 0,Y 432.841,Z 680.59,A -85,B 0,C 180,E1 20315.793,E2 20315.793} C_VEL
LIN {X 0,Y 434.178,Z 662.542,A -85,B 0,C 180,E1 20314.638,E2 20314.638} C_VEL
LIN {X 0,Y 435.304,Z 643.956,A -85,B 0,C 180,E1 20313.719,E2 20313.719} C_VEL
LIN {X 0,Y 436.243,Z 624.097,A -85,B 0,C 180,E1 20313.011,E2 20313.011} C_VEL
LIN {X 0,Y 436.902,Z 602.168,A -85,B 0,C 180,E1 20312.512,E2 20312.512} C_VEL
LIN {X 0,Y 441.546,Z 431.431,A -85,B 0,C 180,E1 20309.188,E2 20309.188} C_VEL
LIN {X 0,Y 437.716,Z 410.777,A -85,B 0,C 180,E1 20308.46,E2 20308.46} C_VEL
LIN {X 0,Y 436.908,Z 408.913,A -85,B 0,C 180,E1 20308.356,E2 20308.356} C_VEL
LIN {X 0,Y 430.163,Z 387.999,A -85,B 0,C 180,E1 20305.604,E2 20305.604} C_VEL
LIN {X 0,Y 425.252,Z 373.828,A -85,B 0,C 180,E1 20303.665,E2 20303.665} C_VEL
LIN {X 0,Y 425.26,Z 373.824,A -85,B 0,C 180,E1 20299.892,E2 20299.892} C_VEL
LIN {X 0,Y 425.287,Z 373.824,A -85,B 0,C 180,E1 20296.201,E2 20296.201} C_VEL
LIN {X 0,Y 425.301,Z 373.823,A -85,B 0,C 180,E1 20292.422,E2 20292.422} C_VEL
LIN {X 0,Y 425.281,Z 373.824,A -85,B 0,C 180,E1 20288.689,E2 20288.689} C_VEL
LIN {X 0,Y 425.256,Z 373.825,A -85,B 0,C 180,E1 20285.008,E2 20285.008} C_VEL
LIN {X 0,Y 425.251,Z 373.825,A -85,B 0,C 180,E1 20281.307,E2 20281.307} C_VEL
LIN {X 0,Y 425.251,Z 373.822,A -85,B 0,C 180,E1 20279.111,E2 20279.111} C_VEL
LIN {X 0,Y 424.267,Z 373.952,A -85,B 0,C 180,E1 20278.073,E2 20278.073} C_VEL
LIN {X 0,Y 417.757,Z 374.762,A -85,B 0,C 180,E1 20275.072,E2 20275.072} C_VEL
LIN {X 0,Y 417.354,Z 374.812,A -85,B 0,C 180,E1 20274.384,E2 20274.384} C_VEL
LIN {X 0,Y 417.331,Z 374.81,A -85,B 0,C 180,E1 20270.621,E2 20270.621} C_VEL
LIN {X 0,Y 417.316,Z 374.809,A -85,B 0,C 180,E1 20266.852,E2 20266.852} C_VEL
LIN {X 0,Y 417.31,Z 374.809,A -85,B 0,C 180,E1 20263.016,E2 20263.016} C_VEL
LIN {X 0,Y 417.31,Z 374.809,A -85,B 0,C 180,E1 20259.099,E2 20259.099} C_VEL
LIN {X 0,Y 417.312,Z 374.811,A -85,B 0,C 180,E1 20255.224,E2 20255.224} C_VEL
LIN {X 0,Y 417.325,Z 374.813,A -85,B 0,C 180,E1 20251.51,E2 20251.51} C_VEL
LIN {X 0,Y 417.352,Z 374.806,A -85,B 0,C 180,E1 20247.803,E2 20247.803} C_VEL
LIN {X 0,Y 417.36,Z 374.81,A -85,B 0,C 180,E1 20243.831,E2 20243.831} C_VEL
LIN {X 0,Y 417.354,Z 374.812,A -85,B 0,C 180,E1 20239.928,E2 20239.928} C_VEL
LIN {X 0,Y 417.351,Z 374.811,A -85,B 0,C 180,E1 20235.995,E2 20235.995} C_VEL
LIN {X 0,Y 417.334,Z 374.811,A -85,B 0,C 180,E1 20232.141,E2 20232.141} C_VEL
LIN {X 0,Y 417.318,Z 374.812,A -85,B 0,C 180,E1 20228.348,E2 20228.348} C_VEL
LIN {X 0,Y 417.31,Z 374.812,A -85,B 0,C 180,E1 20224.593,E2 20224.593} C_VEL
LIN {X 0,Y 417.309,Z 374.812,A -85,B 0,C 180,E1 20220.708,E2 20220.708} C_VEL
LIN {X 0,Y 417.312,Z 374.816,A -85,B 0,C 180,E1 20216.888,E2 20216.888} C_VEL
LIN {X 0,Y 417.331,Z 374.817,A -85,B 0,C 180,E1 20213.151,E2 20213.151} C_VEL
LIN {X 0,Y 417.358,Z 374.814,A -85,B 0,C 180,E1 20209.415,E2 20209.415} C_VEL
LIN {X 0,Y 417.353,Z 374.812,A -85,B 0,C 180,E1 20205.555,E2 20205.555} C_VEL
LIN {X 0,Y 417.349,Z 374.813,A -85,B 0,C 180,E1 20201.628,E2 20201.628} C_VEL
LIN {X 0,Y 417.316,Z 374.817,A -85,B 0,C 180,E1 20197.976,E2 20197.976} C_VEL
LIN {X 0,Y 417.351,Z 374.839,A -85,B 0,C 180,E1 20195.533,E2 20195.533} C_VEL
LIN {X 0,Y 422.929,Z 395.072,A -85,B 0,C 180,E1 20191.926,E2 20191.926} C_VEL
LIN {X 0,Y 425.905,Z 407.347,A -85,B 0,C 180,E1 20189.848,E2 20189.848} C_VEL
LIN {X 0,Y 423.838,Z 434.243,A -85,B 0,C 180,E1 20185.998,E2 20185.998} C_VEL
LIN {X 0,Y 421.815,Z 463.116,A -85,B 0,C 180,E1 20181.922,E2 20181.922} C_VEL
LIN {X 0,Y 420.889,Z 479.164,A -85,B 0,C 180,E1 20179.724,E2 20179.724} C_VEL
LIN {X 0,Y 424.075,Z 502.624,A -85,B 0,C 180,E1 20179.025,E2 20179.025} C_VEL
LIN {X 0,Y 421.682,Z 602.511,A -85,B 0,C 180,E1 20176.846,E2 20176.846} C_VEL
LIN {X 0,Y 421.282,Z 618.038,A -85,B 0,C 180,E1 20176.264,E2 20176.264} C_VEL
LIN {X 0,Y 420.736,Z 633.331,A -85,B 0,C 180,E1 20175.436,E2 20175.436} C_VEL
LIN {X 0,Y 420.022,Z 648.366,A -85,B 0,C 180,E1 20174.334,E2 20174.334} C_VEL
LIN {X 0,Y 419.36,Z 661.43,A -85,B 0,C 180,E1 20173.092,E2 20173.092} C_VEL
LIN {X 0,Y 418.764,Z 673.018,A -85,B 0,C 180,E1 20171.71,E2 20171.71} C_VEL
LIN {X 0,Y 418.177,Z 684.03,A -85,B 0,C 180,E1 20170.052,E2 20170.052} C_VEL
LIN {X 0,Y 417.719,Z 693.315,A -85,B 0,C 180,E1 20168.257,E2 20168.257} C_VEL
LIN {X 0,Y 417.413,Z 700.473,A -85,B 0,C 180,E1 20166.464,E2 20166.464} C_VEL
LIN {X 0,Y 417.228,Z 706.277,A -85,B 0,C 180,E1 20164.496,E2 20164.496} C_VEL
LIN {X 0,Y 417.154,Z 710.206,A -85,B 0,C 180,E1 20162.473,E2 20162.473} C_VEL
LIN {X 0,Y 417.205,Z 712.261,A -85,B 0,C 180,E1 20160.549,E2 20160.549} C_VEL
LIN {X 0,Y 417.319,Z 712.577,A -85,B 0,C 180,E1 20158.49,E2 20158.49} C_VEL
LIN {X 0,Y 417.543,Z 711.166,A -85,B 0,C 180,E1 20156.568,E2 20156.568} C_VEL
LIN {X 0,Y 417.906,Z 707.609,A -85,B 0,C 180,E1 20154.446,E2 20154.446} C_VEL
LIN {X 0,Y 418.422,Z 702.178,A -85,B 0,C 180,E1 20152.448,E2 20152.448} C_VEL
LIN {X 0,Y 419.026,Z 695.442,A -85,B 0,C 180,E1 20150.662,E2 20150.662} C_VEL
LIN {X 0,Y 419.805,Z 686.535,A -85,B 0,C 180,E1 20148.877,E2 20148.877} C_VEL
LIN {X 0,Y 420.7,Z 675.905,A -85,B 0,C 180,E1 20147.231,E2 20147.231} C_VEL
LIN {X 0,Y 421.62,Z 664.184,A -85,B 0,C 180,E1 20145.792,E2 20145.792} C_VEL
LIN {X 0,Y 422.587,Z 650.725,A -85,B 0,C 180,E1 20144.493,E2 20144.493} C_VEL
LIN {X 0,Y 423.522,Z 636.04,A -85,B 0,C 180,E1 20143.402,E2 20143.402} C_VEL
LIN {X 0,Y 424.384,Z 619.551,A -85,B 0,C 180,E1 20142.484,E2 20142.484} C_VEL
LIN {X 0,Y 425.065,Z 602.562,A -85,B 0,C 180,E1 20141.831,E2 20141.831} C_VEL
LIN {X 0,Y 430.111,Z 516.624,A -85,B 0,C 180,E1 20139.317,E2 20139.317} C_VEL
LIN {X 0,Y 430.753,Z 504.585,A -85,B 0,C 180,E1 20138.945,E2 20138.945} C_VEL
LIN {X 0,Y 427.449,Z 484.791,A -85,B 0,C 180,E1 20137.865,E2 20137.865} C_VEL
LIN {X 0,Y 426.282,Z 478.75,A -85,B 0,C 180,E1 20137.486,E2 20137.486} C_VEL
LIN {X 0,Y 429.722,Z 453.087,A -85,B 0,C 180,E1 20133.466,E2 20133.466} C_VEL
LIN {X 0,Y 434.104,Z 428.561,A -85,B 0,C 180,E1 20129.401,E2 20129.401} C_VEL
LIN {X 0,Y 435.235,Z 423,A -85,B 0,C 180,E1 20128.414,E2 20128.414} C_VEL
LIN {X 0,Y 433.622,Z 414.51,A -85,B 0,C 180,E1 20126.109,E2 20126.109} C_VEL
LIN {X 0,Y 431.999,Z 407.925,A -85,B 0,C 180,E1 20123.829,E2 20123.829} C_VEL
LIN {X 0,Y 430.768,Z 403.821,A -85,B 0,C 180,E1 20121.873,E2 20121.873} C_VEL
LIN {X 0,Y 430.161,Z 401.624,A -85,B 0,C 180,E1 20120.441,E2 20120.441} C_VEL
LIN {X 0,Y 429.768,Z 399.473,A -85,B 0,C 180,E1 20117.916,E2 20117.916} C_VEL
LIN {X 0,Y 429.992,Z 399.491,A -85,B 0,C 180,E1 20116.124,E2 20116.124} C_VEL
LIN {X 0,Y 430.657,Z 401.874,A -85,B 0,C 180,E1 20113.776,E2 20113.776} C_VEL
LIN {X 0,Y 431.638,Z 403.696,A -85,B 0,C 180,E1 20112.556,E2 20112.556} C_VEL
LIN {X 0,Y 433.221,Z 408.105,A -85,B 0,C 180,E1 20110.697,E2 20110.697} C_VEL
LIN {X 0,Y 434.974,Z 412.995,A -85,B 0,C 180,E1 20109.123,E2 20109.123} C_VEL
LIN {X 0,Y 437.216,Z 420.51,A -85,B 0,C 180,E1 20107.266,E2 20107.266} C_VEL
LIN {X 0,Y 438.239,Z 425.017,A -85,B 0,C 180,E1 20106.353,E2 20106.353} C_VEL
LIN {X 0,Y 433.273,Z 449.452,A -85,B 0,C 180,E1 20103.473,E2 20103.473} C_VEL
LIN {X 0,Y 430.751,Z 466.671,A -85,B 0,C 180,E1 20101.609,E2 20101.609} C_VEL
LIN {X 0,Y 433.217,Z 488.852,A -85,B 0,C 180,E1 20100.928,E2 20100.928} C_VEL
LIN {X 0,Y 427.989,Z 668.68,A -85,B 0,C 180,E1 20097.292,E2 20097.292} C_VEL
LIN {X 0,Y 426.961,Z 687.994,A -85,B 0,C 180,E1 20096.659,E2 20096.659} C_VEL
LIN {X 0,Y 425.741,Z 706.04,A -85,B 0,C 180,E1 20095.827,E2 20095.827} C_VEL
LIN {X 0,Y 424.306,Z 724.218,A -85,B 0,C 180,E1 20094.726,E2 20094.726} C_VEL
LIN {X 0,Y 422.825,Z 741.409,A -85,B 0,C 180,E1 20093.408,E2 20093.408} C_VEL
LIN {X 0,Y 421.344,Z 757.639,A -85,B 0,C 180,E1 20091.874,E2 20091.874} C_VEL
LIN {X 0,Y 419.962,Z 772.596,A -85,B 0,C 180,E1 20090.155,E2 20090.155} C_VEL
LIN {X 0,Y 418.725,Z 786.43,A -85,B 0,C 180,E1 20088.229,E2 20088.229} C_VEL
LIN {X 0,Y 417.682,Z 798.88,A -85,B 0,C 180,E1 20086.122,E2 20086.122} C_VEL
LIN {X 0,Y 416.939,Z 809.756,A -85,B 0,C 180,E1 20083.875,E2 20083.875} C_VEL
LIN {X 0,Y 416.454,Z 818.655,A -85,B 0,C 180,E1 20081.604,E2 20081.604} C_VEL
LIN {X 0,Y 416.218,Z 825.904,A -85,B 0,C 180,E1 20079.262,E2 20079.262} C_VEL
LIN {X 0,Y 416.151,Z 831.429,A -85,B 0,C 180,E1 20076.9,E2 20076.9} C_VEL
LIN {X 0,Y 416.156,Z 835.257,A -85,B 0,C 180,E1 20074.548,E2 20074.548} C_VEL
LIN {X 0,Y 416.199,Z 837.477,A -85,B 0,C 180,E1 20072.203,E2 20072.203} C_VEL
LIN {X 0,Y 416.228,Z 838.13,A -85,B 0,C 180,E1 20069.862,E2 20069.862} C_VEL
LIN {X 0,Y 416.198,Z 837.094,A -85,B 0,C 180,E1 20067.384,E2 20067.384} C_VEL
LIN {X 0,Y 416.165,Z 834.286,A -85,B 0,C 180,E1 20064.9,E2 20064.9} C_VEL
LIN {X 0,Y 416.164,Z 829.64,A -85,B 0,C 180,E1 20062.407,E2 20062.407} C_VEL
LIN {X 0,Y 416.269,Z 823.323,A -85,B 0,C 180,E1 20059.998,E2 20059.998} C_VEL
LIN {X 0,Y 416.581,Z 815.317,A -85,B 0,C 180,E1 20057.651,E2 20057.651} C_VEL
LIN {X 0,Y 417.104,Z 805.807,A -85,B 0,C 180,E1 20055.422,E2 20055.422} C_VEL
LIN {X 0,Y 417.88,Z 794.837,A -85,B 0,C 180,E1 20053.314,E2 20053.314} C_VEL
LIN {X 0,Y 418.934,Z 782.032,A -85,B 0,C 180,E1 20051.276,E2 20051.276} C_VEL
LIN {X 0,Y 420.268,Z 767.091,A -85,B 0,C 180,E1 20049.311,E2 20049.311} C_VEL
LIN {X 0,Y 421.775,Z 750.97,A -85,B 0,C 180,E1 20047.563,E2 20047.563} C_VEL
LIN {X 0,Y 423.371,Z 733.747,A -85,B 0,C 180,E1 20046.033,E2 20046.033} C_VEL
LIN {X 0,Y 425.002,Z 715.452,A -85,B 0,C 180,E1 20044.723,E2 20044.723} C_VEL
LIN {X 0,Y 426.554,Z 696.589,A -85,B 0,C 180,E1 20043.665,E2 20043.665} C_VEL
LIN {X 0,Y 427.996,Z 676.715,A -85,B 0,C 180,E1 20042.829,E2 20042.829} C_VEL
LIN {X 0,Y 429.17,Z 655.531,A -85,B 0,C 180,E1 20042.212,E2 20042.212} C_VEL
LIN {X 0,Y 432.917,Z 568.447,A -85,B 0,C 180,E1 20040.179,E2 20040.179} C_VEL
LIN {X 0,Y 437.65,Z 487.45,A -85,B 0,C 180,E1 20038.103,E2 20038.103} C_VEL
LIN {X 0,Y 435.861,Z 459.652,A -85,B 0,C 180,E1 20036.866,E2 20036.866} C_VEL
LIN {X 0,Y 434.16,Z 436.346,A -85,B 0,C 180,E1 20035.621,E2 20035.621} C_VEL
LIN {X 0,Y 433.277,Z 418.62,A -85,B 0,C 180,E1 20034.451,E2 20034.451} C_VEL
LIN {X 0,Y 429.216,Z 406.022,A -85,B 0,C 180,E1 20032.692,E2 20032.692} C_VEL
LIN {X 0,Y 426.528,Z 393.769,A -85,B 0,C 180,E1 20030.676,E2 20030.676} C_VEL
LIN {X 0,Y 425.376,Z 386.579,A -85,B 0,C 180,E1 20029.086,E2 20029.086} C_VEL
LIN {X 0,Y 423.295,Z 384.29,A -85,B 0,C 180,E1 20026.877,E2 20026.877} C_VEL
LIN {X 0,Y 422.968,Z 383.841,A -85,B 0,C 180,E1 20025.168,E2 20025.168} C_VEL
LIN {X 0,Y 423.788,Z 385.35,A -85,B 0,C 180,E1 20022.988,E2 20022.988} C_VEL
LIN {X 0,Y 425.421,Z 386.915,A -85,B 0,C 180,E1 20021.512,E2 20021.512} C_VEL
LIN {X 0,Y 426.734,Z 390.348,A -85,B 0,C 180,E1 20020.196,E2 20020.196} C_VEL
LIN {X 0,Y 427.918,Z 392.056,A -85,B 0,C 180,E1 20019.46,E2 20019.46} C_VEL
LIN {X 0,Y 430.273,Z 397.292,A -85,B 0,C 180,E1 20017.915,E2 20017.915} C_VEL
LIN {X 0,Y 432.801,Z 402.974,A -85,B 0,C 180,E1 20016.49,E2 20016.49} C_VEL
LIN {X 0,Y 436.008,Z 412.524,A -85,B 0,C 180,E1 20014.587,E2 20014.587} C_VEL
LIN {X 0,Y 437.993,Z 419.342,A -85,B 0,C 180,E1 20013.479,E2 20013.479} C_VEL
LIN {X 0,Y 439.579,Z 423.403,A -85,B 0,C 180,E1 20013.064,E2 20013.064} C_VEL
LIN {X 0,Y 441.089,Z 436.057,A -85,B 0,C 180,E1 20012.363,E2 20012.363} C_VEL
LIN {X 0,Y 434.801,Z 527.549,A -85,B 0,C 180,E1 20010.001,E2 20010.001} C_VEL
LIN {X 0,Y 430.875,Z 609.08,A -85,B 0,C 180,E1 20008.066,E2 20008.066} C_VEL
LIN {X 0,Y 429.919,Z 631.7,A -85,B 0,C 180,E1 20007.451,E2 20007.451} C_VEL
LIN {X 0,Y 428.821,Z 651.018,A -85,B 0,C 180,E1 20006.669,E2 20006.669} C_VEL
LIN {X 0,Y 427.535,Z 668.749,A -85,B 0,C 180,E1 20005.71,E2 20005.71} C_VEL
LIN {X 0,Y 426,Z 686.613,A -85,B 0,C 180,E1 20004.473,E2 20004.473} C_VEL
LIN {X 0,Y 424.386,Z 703.385,A -85,B 0,C 180,E1 20003.023,E2 20003.023} C_VEL
LIN {X 0,Y 422.749,Z 719.073,A -85,B 0,C 180,E1 20001.36,E2 20001.36} C_VEL
LIN {X 0,Y 421.209,Z 733.199,A -85,B 0,C 180,E1 19999.542,E2 19999.542} C_VEL
LIN {X 0,Y 419.844,Z 745.654,A -85,B 0,C 180,E1 19997.605,E2 19997.605} C_VEL
LIN {X 0,Y 418.667,Z 756.759,A -85,B 0,C 180,E1 19995.514,E2 19995.514} C_VEL
LIN {X 0,Y 417.716,Z 766.423,A -85,B 0,C 180,E1 19993.284,E2 19993.284} C_VEL
LIN {X 0,Y 417.003,Z 774.599,A -85,B 0,C 180,E1 19990.919,E2 19990.919} C_VEL
LIN {X 0,Y 416.522,Z 781.194,A -85,B 0,C 180,E1 19988.42,E2 19988.42} C_VEL
LIN {X 0,Y 416.252,Z 785.908,A -85,B 0,C 180,E1 19985.928,E2 19985.928} C_VEL
LIN {X 0,Y 416.122,Z 788.879,A -85,B 0,C 180,E1 19983.444,E2 19983.444} C_VEL
LIN {X 0,Y 416.07,Z 790.18,A -85,B 0,C 180,E1 19980.964,E2 19980.964} C_VEL
LIN {X 0,Y 416.058,Z 789.831,A -85,B 0,C 180,E1 19978.485,E2 19978.485} C_VEL
LIN {X 0,Y 416.092,Z 787.834,A -85,B 0,C 180,E1 19976.004,E2 19976.004} C_VEL
LIN {X 0,Y 416.209,Z 784.14,A -85,B 0,C 180,E1 19973.517,E2 19973.517} C_VEL
LIN {X 0,Y 416.462,Z 778.651,A -85,B 0,C 180,E1 19971.022,E2 19971.022} C_VEL
LIN {X 0,Y 416.925,Z 771.217,A -85,B 0,C 180,E1 19968.518,E2 19968.518} C_VEL
LIN {X 0,Y 417.626,Z 762.184,A -85,B 0,C 180,E1 19966.148,E2 19966.148} C_VEL
LIN {X 0,Y 418.567,Z 751.603,A -85,B 0,C 180,E1 19963.913,E2 19963.913} C_VEL
LIN {X 0,Y 419.741,Z 739.491,A -85,B 0,C 180,E1 19961.817,E2 19961.817} C_VEL
LIN {X 0,Y 421.103,Z 725.77,A -85,B 0,C 180,E1 19959.862,E2 19959.862} C_VEL
LIN {X 0,Y 422.562,Z 710.94,A -85,B 0,C 180,E1 19958.119,E2 19958.119} C_VEL
LIN {X 0,Y 424.034,Z 695.154,A -85,B 0,C 180,E1 19956.589,E2 19956.589} C_VEL
LIN {X 0,Y 425.53,Z 677.754,A -85,B 0,C 180,E1 19955.219,E2 19955.219} C_VEL
LIN {X 0,Y 426.918,Z 659.395,A -85,B 0,C 180,E1 19954.073,E2 19954.073} C_VEL
LIN {X 0,Y 428.04,Z 641.223,A -85,B 0,C 180,E1 19953.203,E2 19953.203} C_VEL
LIN {X 0,Y 428.951,Z 621.82,A -85,B 0,C 180,E1 19952.533,E2 19952.533} C_VEL
LIN {X 0,Y 429.743,Z 594.009,A -85,B 0,C 180,E1 19951.936,E2 19951.936} C_VEL
LIN {X 0,Y 434.439,Z 432.496,A -85,B 0,C 180,E1 19948.709,E2 19948.709} C_VEL
LIN {X 0,Y 431.003,Z 413.865,A -85,B 0,C 180,E1 19948.032,E2 19948.032} C_VEL
LIN {X 0,Y 428.799,Z 409.001,A -85,B 0,C 180,E1 19947.725,E2 19947.725} C_VEL
LIN {X 0,Y 421.596,Z 387.246,A -85,B 0,C 180,E1 19944.809,E2 19944.809} C_VEL
LIN {X 0,Y 417.327,Z 374.814,A -85,B 0,C 180,E1 19943.079,E2 19943.079} C_VEL
LIN {X 0,Y 417.314,Z 374.815,A -85,B 0,C 180,E1 19939.33,E2 19939.33} C_VEL
LIN {X 0,Y 417.314,Z 374.815,A -85,B 0,C 180,E1 19935.561,E2 19935.561} C_VEL
LIN {X 0,Y 417.321,Z 374.812,A -85,B 0,C 180,E1 19931.764,E2 19931.764} C_VEL
LIN {X 0,Y 417.353,Z 374.812,A -85,B 0,C 180,E1 19928.177,E2 19928.177} C_VEL
LIN {X 0,Y 417.355,Z 374.813,A -85,B 0,C 180,E1 19924.257,E2 19924.257} C_VEL
LIN {X 0,Y 417.366,Z 374.813,A -85,B 0,C 180,E1 19920.363,E2 19920.363} C_VEL
LIN {X 0,Y 417.348,Z 374.811,A -85,B 0,C 180,E1 19916.462,E2 19916.462} C_VEL
LIN {X 0,Y 417.354,Z 374.812,A -85,B 0,C 180,E1 19914.384,E2 19914.384} C_VEL
LIN {X 0,Y 416.414,Z 374.929,A -85,B 0,C 180,E1 19913.327,E2 19913.327} C_VEL
LIN {X 0,Y 411.642,Z 375.527,A -85,B 0,C 180,E1 19911.259,E2 19911.259} C_VEL
LIN {X 0,Y 409.544,Z 375.786,A -85,B 0,C 180,E1 19909.961,E2 19909.961} C_VEL
LIN {X 0,Y 409.383,Z 375.802,A -85,B 0,C 180,E1 19909.57,E2 19909.57} C_VEL
LIN {X 0,Y 409.394,Z 375.803,A -85,B 0,C 180,E1 19905.729,E2 19905.729} C_VEL
LIN {X 0,Y 409.415,Z 375.801,A -85,B 0,C 180,E1 19901.981,E2 19901.981} C_VEL
LIN {X 0,Y 409.425,Z 375.796,A -85,B 0,C 180,E1 19898.002,E2 19898.002} C_VEL
LIN {X 0,Y 409.414,Z 375.796,A -85,B 0,C 180,E1 19894.061,E2 19894.061} C_VEL
LIN {X 0,Y 409.412,Z 375.801,A -85,B 0,C 180,E1 19890.14,E2 19890.14} C_VEL
LIN {X 0,Y 409.399,Z 375.798,A -85,B 0,C 180,E1 19886.219,E2 19886.219} C_VEL
LIN {X 0,Y 409.384,Z 375.797,A -85,B 0,C 180,E1 19882.421,E2 19882.421} C_VEL
LIN {X 0,Y 409.374,Z 375.801,A -85,B 0,C 180,E1 19878.59,E2 19878.59} C_VEL
LIN {X 0,Y 409.37,Z 375.803,A -85,B 0,C 180,E1 19874.746,E2 19874.746} C_VEL
LIN {X 0,Y 409.373,Z 375.803,A -85,B 0,C 180,E1 19870.896,E2 19870.896} C_VEL
LIN {X 0,Y 409.377,Z 375.801,A -85,B 0,C 180,E1 19867.041,E2 19867.041} C_VEL
LIN {X 0,Y 409.395,Z 375.801,A -85,B 0,C 180,E1 19863.296,E2 19863.296} C_VEL
LIN {X 0,Y 409.414,Z 375.804,A -85,B 0,C 180,E1 19859.471,E2 19859.471} C_VEL
LIN {X 0,Y 409.415,Z 375.804,A -85,B 0,C 180,E1 19855.487,E2 19855.487} C_VEL
LIN {X 0,Y 409.424,Z 375.803,A -85,B 0,C 180,E1 19851.483,E2 19851.483} C_VEL
LIN {X 0,Y 409.417,Z 375.802,A -85,B 0,C 180,E1 19847.522,E2 19847.522} C_VEL
LIN {X 0,Y 409.414,Z 375.802,A -85,B 0,C 180,E1 19843.527,E2 19843.527} C_VEL
LIN {X 0,Y 409.401,Z 375.805,A -85,B 0,C 180,E1 19839.708,E2 19839.708} C_VEL
LIN {X 0,Y 409.383,Z 375.867,A -85,B 0,C 180,E1 19836.058,E2 19836.058} C_VEL
LIN {X 0,Y 414.853,Z 395.464,A -85,B 0,C 180,E1 19832.482,E2 19832.482} C_VEL
LIN {X 0,Y 418.339,Z 409.275,A -85,B 0,C 180,E1 19830.093,E2 19830.093} C_VEL
LIN {X 0,Y 416.15,Z 436.254,A -85,B 0,C 180,E1 19826.171,E2 19826.171} C_VEL
LIN {X 0,Y 414.044,Z 465.006,A -85,B 0,C 180,E1 19822.056,E2 19822.056} C_VEL
LIN {X 0,Y 413.203,Z 479.041,A -85,B 0,C 180,E1 19820.113,E2 19820.113} C_VEL
LIN {X 0,Y 416.5,Z 503.459,A -85,B 0,C 180,E1 19819.368,E2 19819.368} C_VEL
LIN {X 0,Y 413.961,Z 602.86,A -85,B 0,C 180,E1 19817.129,E2 19817.129} C_VEL
LIN {X 0,Y 413.545,Z 618.32,A -85,B 0,C 180,E1 19816.541,E2 19816.541} C_VEL
LIN {X 0,Y 412.949,Z 634.236,A -85,B 0,C 180,E1 19815.663,E2 19815.663} C_VEL
LIN {X 0,Y 412.164,Z 650.078,A -85,B 0,C 180,E1 19814.47,E2 19814.47} C_VEL
LIN {X 0,Y 411.427,Z 664.266,A -85,B 0,C 180,E1 19813.063,E2 19813.063} C_VEL
LIN {X 0,Y 410.753,Z 676.445,A -85,B 0,C 180,E1 19811.514,E2 19811.514} C_VEL
LIN {X 0,Y 410.222,Z 686.186,A -85,B 0,C 180,E1 19809.966,E2 19809.966} C_VEL
LIN {X 0,Y 409.767,Z 695.307,A -85,B 0,C 180,E1 19808.136,E2 19808.136} C_VEL
LIN {X 0,Y 409.452,Z 702.726,A -85,B 0,C 180,E1 19806.168,E2 19806.168} C_VEL
LIN {X 0,Y 409.292,Z 707.82,A -85,B 0,C 180,E1 19804.343,E2 19804.343} C_VEL
LIN {X 0,Y 409.246,Z 711.796,A -85,B 0,C 180,E1 19802.198,E2 19802.198} C_VEL
LIN {X 0,Y 409.3,Z 713.667,A -85,B 0,C 180,E1 19800.14,E2 19800.14} C_VEL
LIN {X 0,Y 409.466,Z 713.797,A -85,B 0,C 180,E1 19798.181,E2 19798.181} C_VEL
LIN {X 0,Y 409.737,Z 712.028,A -85,B 0,C 180,E1 19796.082,E2 19796.082} C_VEL
LIN {X 0,Y 410.136,Z 708.626,A -85,B 0,C 180,E1 19794.123,E2 19794.123} C_VEL
LIN {X 0,Y 410.741,Z 702.872,A -85,B 0,C 180,E1 19792.024,E2 19792.024} C_VEL
LIN {X 0,Y 411.415,Z 695.88,A -85,B 0,C 180,E1 19790.205,E2 19790.205} C_VEL
LIN {X 0,Y 412.266,Z 687.253,A -85,B 0,C 180,E1 19788.469,E2 19788.469} C_VEL
LIN {X 0,Y 413.216,Z 676.924,A -85,B 0,C 180,E1 19786.853,E2 19786.853} C_VEL
LIN {X 0,Y 414.206,Z 665.104,A -85,B 0,C 180,E1 19785.389,E2 19785.389} C_VEL
LIN {X 0,Y 415.263,Z 651.673,A -85,B 0,C 180,E1 19784.069,E2 19784.069} C_VEL
LIN {X 0,Y 416.34,Z 636.301,A -85,B 0,C 180,E1 19782.906,E2 19782.906} C_VEL
LIN {X 0,Y 417.249,Z 620.076,A -85,B 0,C 180,E1 19781.994,E2 19781.994} C_VEL
LIN {X 0,Y 418.048,Z 601.646,A -85,B 0,C 180,E1 19781.282,E2 19781.282} C_VEL
LIN {X 0,Y 424.19,Z 506.091,A -85,B 0,C 180,E1 19778.353,E2 19778.353} C_VEL
LIN {X 0,Y 421.125,Z 486.932,A -85,B 0,C 180,E1 19777.25,E2 19777.25} C_VEL
LIN {X 0,Y 419.536,Z 478.572,A -85,B 0,C 180,E1 19776.696,E2 19776.696} C_VEL
LIN {X 0,Y 423.403,Z 453.045,A -85,B 0,C 180,E1 19772.581,E2 19772.581} C_VEL
LIN {X 0,Y 427.893,Z 430.711,A -85,B 0,C 180,E1 19768.752,E2 19768.752} C_VEL
LIN {X 0,Y 428.737,Z 426.847,A -85,B 0,C 180,E1 19768.036,E2 19768.036} C_VEL
LIN {X 0,Y 427.378,Z 419.146,A -85,B 0,C 180,E1 19765.842,E2 19765.842} C_VEL
LIN {X 0,Y 426.042,Z 412.952,A -85,B 0,C 180,E1 19763.576,E2 19763.576} C_VEL
LIN {X 0,Y 424.922,Z 408.788,A -85,B 0,C 180,E1 19761.424,E2 19761.424} C_VEL
LIN {X 0,Y 424.46,Z 407.087,A -85,B 0,C 180,E1 19760.154,E2 19760.154} C_VEL
LIN {X 0,Y 424.377,Z 405.195,A -85,B 0,C 180,E1 19757.454,E2 19757.454} C_VEL
LIN {X 0,Y 424.593,Z 405.539,A -85,B 0,C 180,E1 19755.909,E2 19755.909} C_VEL
LIN {X 0,Y 425.491,Z 408.222,A -85,B 0,C 180,E1 19753.438,E2 19753.438} C_VEL
LIN {X 0,Y 426.162,Z 409.783,A -85,B 0,C 180,E1 19752.509,E2 19752.509} C_VEL
LIN {X 0,Y 427.648,Z 413.965,A -85,B 0,C 180,E1 19750.717,E2 19750.717} C_VEL
LIN {X 0,Y 429.732,Z 420.231,A -85,B 0,C 180,E1 19748.747,E2 19748.747} C_VEL
LIN {X 0,Y 431.793,Z 428.302,A -85,B 0,C 180,E1 19746.852,E2 19746.852} C_VEL
LIN {X 0,Y 426.881,Z 450.595,A -85,B 0,C 180,E1 19744.123,E2 19744.123} C_VEL
LIN {X 0,Y 423.93,Z 468.429,A -85,B 0,C 180,E1 19742.118,E2 19742.118} C_VEL
LIN {X 0,Y 426.083,Z 487.882,A -85,B 0,C 180,E1 19741.457,E2 19741.457} C_VEL
LIN {X 0,Y 420.583,Z 668.318,A -85,B 0,C 180,E1 19737.705,E2 19737.705} C_VEL
LIN {X 0,Y 419.506,Z 687.605,A -85,B 0,C 180,E1 19737.061,E2 19737.061} C_VEL
LIN {X 0,Y 418.161,Z 706.475,A -85,B 0,C 180,E1 19736.169,E2 19736.169} C_VEL
LIN {X 0,Y 416.677,Z 724.363,A -85,B 0,C 180,E1 19735.058,E2 19735.058} C_VEL
LIN {X 0,Y 415.13,Z 741.451,A -85,B 0,C 180,E1 19733.718,E2 19733.718} C_VEL
LIN {X 0,Y 413.582,Z 757.604,A -85,B 0,C 180,E1 19732.157,E2 19732.157} C_VEL
LIN {X 0,Y 412.111,Z 772.755,A -85,B 0,C 180,E1 19730.375,E2 19730.375} C_VEL
LIN {X 0,Y 410.839,Z 786.293,A -85,B 0,C 180,E1 19728.444,E2 19728.444} C_VEL
LIN {X 0,Y 409.751,Z 798.72,A -85,B 0,C 180,E1 19726.297,E2 19726.297} C_VEL
LIN {X 0,Y 409.012,Z 808.972,A -85,B 0,C 180,E1 19724.15,E2 19724.15} C_VEL
LIN {X 0,Y 408.493,Z 817.856,A -85,B 0,C 180,E1 19721.865,E2 19721.865} C_VEL
LIN {X 0,Y 408.23,Z 825.282,A -85,B 0,C 180,E1 19719.445,E2 19719.445} C_VEL
LIN {X 0,Y 408.162,Z 830.866,A -85,B 0,C 180,E1 19717.035,E2 19717.035} C_VEL
LIN {X 0,Y 408.165,Z 834.739,A -85,B 0,C 180,E1 19714.637,E2 19714.637} C_VEL
LIN {X 0,Y 408.211,Z 836.991,A -85,B 0,C 180,E1 19712.246,E2 19712.246} C_VEL
LIN {X 0,Y 408.242,Z 837.659,A -85,B 0,C 180,E1 19709.86,E2 19709.86} C_VEL
LIN {X 0,Y 408.207,Z 836.632,A -85,B 0,C 180,E1 19707.333,E2 19707.333} C_VEL
LIN {X 0,Y 408.167,Z 833.825,A -85,B 0,C 180,E1 19704.8,E2 19704.8} C_VEL
LIN {X 0,Y 408.166,Z 829.173,A -85,B 0,C 180,E1 19702.257,E2 19702.257} C_VEL
LIN {X 0,Y 408.282,Z 822.983,A -85,B 0,C 180,E1 19699.844,E2 19699.844} C_VEL
LIN {X 0,Y 408.625,Z 814.886,A -85,B 0,C 180,E1 19697.422,E2 19697.422} C_VEL
LIN {X 0,Y 409.204,Z 805.31,A -85,B 0,C 180,E1 19695.134,E2 19695.134} C_VEL
LIN {X 0,Y 410.096,Z 793.779,A -85,B 0,C 180,E1 19692.889,E2 19692.889} C_VEL
LIN {X 0,Y 411.242,Z 781.041,A -85,B 0,C 180,E1 19690.839,E2 19690.839} C_VEL
LIN {X 0,Y 412.665,Z 766.373,A -85,B 0,C 180,E1 19688.88,E2 19688.88} C_VEL
LIN {X 0,Y 414.264,Z 750.562,A -85,B 0,C 180,E1 19687.133,E2 19687.133} C_VEL
LIN {X 0,Y 415.98,Z 733.449,A -85,B 0,C 180,E1 19685.58,E2 19685.58} C_VEL
LIN {X 0,Y 417.731,Z 715.367,A -85,B 0,C 180,E1 19684.251,E2 19684.251} C_VEL
LIN {X 0,Y 419.443,Z 696.16,A -85,B 0,C 180,E1 19683.145,E2 19683.145} C_VEL
LIN {X 0,Y 421.013,Z 676.433,A -85,B 0,C 180,E1 19682.292,E2 19682.292} C_VEL
LIN {X 0,Y 422.322,Z 655.086,A -85,B 0,C 180,E1 19681.646,E2 19681.646} C_VEL
LIN {X 0,Y 426.234,Z 573.564,A -85,B 0,C 180,E1 19679.663,E2 19679.663} C_VEL
LIN {X 0,Y 431.76,Z 489.197,A -85,B 0,C 180,E1 19677.428,E2 19677.428} C_VEL
LIN {X 0,Y 430.351,Z 461.849,A -85,B 0,C 180,E1 19676.154,E2 19676.154} C_VEL
LIN {X 0,Y 428.948,Z 438.875,A -85,B 0,C 180,E1 19674.885,E2 19674.885} C_VEL
LIN {X 0,Y 428.443,Z 422.931,A -85,B 0,C 180,E1 19673.798,E2 19673.798} C_VEL
LIN {X 0,Y 424.653,Z 409.685,A -85,B 0,C 180,E1 19671.851,E2 19671.851} C_VEL
LIN {X 0,Y 422.73,Z 398.849,A -85,B 0,C 180,E1 19669.958,E2 19669.958} C_VEL
LIN {X 0,Y 422.146,Z 393.779,A -85,B 0,C 180,E1 19668.818,E2 19668.818} C_VEL
LIN {X 0,Y 420.247,Z 391.635,A -85,B 0,C 180,E1 19666.722,E2 19666.722} C_VEL
LIN {X 0,Y 419.839,Z 391.259,A -85,B 0,C 180,E1 19665.017,E2 19665.017} C_VEL
LIN {X 0,Y 420.633,Z 392.895,A -85,B 0,C 180,E1 19662.734,E2 19662.734} C_VEL
LIN {X 0,Y 421.69,Z 394.016,A -85,B 0,C 180,E1 19661.678,E2 19661.678} C_VEL
LIN {X 0,Y 423.085,Z 397.587,A -85,B 0,C 180,E1 19660.178,E2 19660.178} C_VEL
LIN {X 0,Y 423.863,Z 399.167,A -85,B 0,C 180,E1 19659.562,E2 19659.562} C_VEL
LIN {X 0,Y 425.714,Z 403.456,A -85,B 0,C 180,E1 19658.221,E2 19658.221} C_VEL
LIN {X 0,Y 428.102,Z 409.577,A -85,B 0,C 180,E1 19656.653,E2 19656.653} C_VEL
LIN {X 0,Y 430.845,Z 418.298,A -85,B 0,C 180,E1 19654.866,E2 19654.866} C_VEL
LIN {X 0,Y 431.843,Z 421.072,A -85,B 0,C 180,E1 19654.424,E2 19654.424} C_VEL
LIN {X 0,Y 434.507,Z 427.672,A -85,B 0,C 180,E1 19653.672,E2 19653.672} C_VEL
LIN {X 0,Y 435.492,Z 437.922,A -85,B 0,C 180,E1 19653.086,E2 19653.086} C_VEL
LIN {X 0,Y 428.645,Z 527.395,A -85,B 0,C 180,E1 19650.686,E2 19650.686} C_VEL
LIN {X 0,Y 424.376,Z 604.656,A -85,B 0,C 180,E1 19648.761,E2 19648.761} C_VEL
LIN {X 0,Y 423.263,Z 629.277,A -85,B 0,C 180,E1 19648.107,E2 19648.107} C_VEL
LIN {X 0,Y 422.104,Z 648.336,A -85,B 0,C 180,E1 19647.357,E2 19647.357} C_VEL
LIN {X 0,Y 420.678,Z 667.137,A -85,B 0,C 180,E1 19646.356,E2 19646.356} C_VEL
LIN {X 0,Y 419.067,Z 685.043,A -85,B 0,C 180,E1 19645.131,E2 19645.131} C_VEL
LIN {X 0,Y 417.395,Z 701.47,A -85,B 0,C 180,E1 19643.731,E2 19643.731} C_VEL
LIN {X 0,Y 415.674,Z 716.935,A -85,B 0,C 180,E1 19642.113,E2 19642.113} C_VEL
LIN {X 0,Y 413.979,Z 731.391,A -85,B 0,C 180,E1 19640.279,E2 19640.279} C_VEL
LIN {X 0,Y 412.397,Z 744.71,A -85,B 0,C 180,E1 19638.226,E2 19638.226} C_VEL
LIN {X 0,Y 411.085,Z 756.064,A -85,B 0,C 180,E1 19636.098,E2 19636.098} C_VEL
LIN {X 0,Y 410.01,Z 765.947,A -85,B 0,C 180,E1 19633.826,E2 19633.826} C_VEL
LIN {X 0,Y 409.194,Z 774.336,A -85,B 0,C 180,E1 19631.415,E2 19631.415} C_VEL
LIN {X 0,Y 408.659,Z 780.821,A -85,B 0,C 180,E1 19629.009,E2 19629.009} C_VEL
LIN {X 0,Y 408.326,Z 785.831,A -85,B 0,C 180,E1 19626.467,E2 19626.467} C_VEL
LIN {X 0,Y 408.161,Z 789.066,A -85,B 0,C 180,E1 19623.933,E2 19623.933} C_VEL
LIN {X 0,Y 408.095,Z 790.608,A -85,B 0,C 180,E1 19621.404,E2 19621.404} C_VEL
LIN {X 0,Y 408.074,Z 790.491,A -85,B 0,C 180,E1 19618.877,E2 19618.877} C_VEL
LIN {X 0,Y 408.099,Z 788.717,A -85,B 0,C 180,E1 19616.348,E2 19616.348} C_VEL
LIN {X 0,Y 408.206,Z 785.25,A -85,B 0,C 180,E1 19613.813,E2 19613.813} C_VEL
LIN {X 0,Y 408.449,Z 779.984,A -85,B 0,C 180,E1 19611.27,E2 19611.27} C_VEL
LIN {X 0,Y 408.878,Z 773.245,A -85,B 0,C 180,E1 19608.861,E2 19608.861} C_VEL
LIN {X 0,Y 409.555,Z 764.574,A -85,B 0,C 180,E1 19606.445,E2 19606.445} C_VEL
LIN {X 0,Y 410.479,Z 754.388,A -85,B 0,C 180,E1 19604.168,E2 19604.168} C_VEL
LIN {X 0,Y 411.636,Z 742.726,A -85,B 0,C 180,E1 19602.032,E2 19602.032} C_VEL
LIN {X 0,Y 413.06,Z 728.994,A -85,B 0,C 180,E1 19599.962,E2 19599.962} C_VEL
LIN {X 0,Y 414.594,Z 714.192,A -85,B 0,C 180,E1 19598.124,E2 19598.124} C_VEL
LIN {X 0,Y 416.17,Z 698.266,A -85,B 0,C 180,E1 19596.495,E2 19596.495} C_VEL
LIN {X 0,Y 417.723,Z 681.277,A -85,B 0,C 180,E1 19595.085,E2 19595.085} C_VEL
LIN {X 0,Y 419.149,Z 663.652,A -85,B 0,C 180,E1 19593.916,E2 19593.916} C_VEL
LIN {X 0,Y 420.358,Z 645.503,A -85,B 0,C 180,E1 19592.979,E2 19592.979} C_VEL
LIN {X 0,Y 421.381,Z 626.043,A -85,B 0,C 180,E1 19592.246,E2 19592.246} C_VEL
LIN {X 0,Y 422.13,Z 604.21,A -85,B 0,C 180,E1 19591.712,E2 19591.712} C_VEL
LIN {X 0,Y 427.406,Z 433.915,A -85,B 0,C 180,E1 19588.229,E2 19588.229} C_VEL
LIN {X 0,Y 424.356,Z 417.132,A -85,B 0,C 180,E1 19587.608,E2 19587.608} C_VEL
LIN {X 0,Y 420.811,Z 409.433,A -85,B 0,C 180,E1 19587.133,E2 19587.133} C_VEL
LIN {X 0,Y 413.434,Z 387.317,A -85,B 0,C 180,E1 19584.113,E2 19584.113} C_VEL
LIN {X 0,Y 409.423,Z 375.795,A -85,B 0,C 180,E1 19582.46,E2 19582.46} C_VEL
LIN {X 0,Y 409.427,Z 375.799,A -85,B 0,C 180,E1 19578.562,E2 19578.562} C_VEL
LIN {X 0,Y 409.408,Z 375.802,A -85,B 0,C 180,E1 19574.697,E2 19574.697} C_VEL
LIN {X 0,Y 409.391,Z 375.801,A -85,B 0,C 180,E1 19570.885,E2 19570.885} C_VEL
LIN {X 0,Y 409.377,Z 375.803,A -85,B 0,C 180,E1 19567.105,E2 19567.105} C_VEL
LIN {X 0,Y 409.373,Z 375.804,A -85,B 0,C 180,E1 19563.336,E2 19563.336} C_VEL
LIN {X 0,Y 409.373,Z 375.801,A -85,B 0,C 180,E1 19559.402,E2 19559.402} C_VEL
LIN {X 0,Y 409.383,Z 375.802,A -85,B 0,C 180,E1 19555.614,E2 19555.614} C_VEL
LIN {X 0,Y 409.396,Z 375.8,A -85,B 0,C 180,E1 19551.791,E2 19551.791} C_VEL
LIN {X 0,Y 409.383,Z 375.802,A -85,B 0,C 180,E1 19549.57,E2 19549.57} C_VEL
LIN {X 0,Y 408.35,Z 375.934,A -85,B 0,C 180,E1 19548.492,E2 19548.492} C_VEL
LIN {X 0,Y 401.842,Z 376.744,A -85,B 0,C 180,E1 19545.373,E2 19545.373} C_VEL
LIN {X 0,Y 401.445,Z 376.792,A -85,B 0,C 180,E1 19544.658,E2 19544.658} C_VEL
LIN {X 0,Y 401.438,Z 376.791,A -85,B 0,C 180,E1 19540.766,E2 19540.766} C_VEL
LIN {X 0,Y 401.435,Z 376.789,A -85,B 0,C 180,E1 19536.866,E2 19536.866} C_VEL
LIN {X 0,Y 401.43,Z 376.786,A -85,B 0,C 180,E1 19532.998,E2 19532.998} C_VEL
LIN {X 0,Y 401.431,Z 376.786,A -85,B 0,C 180,E1 19529.001,E2 19529.001} C_VEL
LIN {X 0,Y 401.431,Z 376.79,A -85,B 0,C 180,E1 19524.999,E2 19524.999} C_VEL
LIN {X 0,Y 401.435,Z 376.789,A -85,B 0,C 180,E1 19521.117,E2 19521.117} C_VEL
LIN {X 0,Y 401.447,Z 376.789,A -85,B 0,C 180,E1 19517.339,E2 19517.339} C_VEL
LIN {X 0,Y 401.463,Z 376.789,A -85,B 0,C 180,E1 19513.505,E2 19513.505} C_VEL
LIN {X 0,Y 401.473,Z 376.789,A -85,B 0,C 180,E1 19509.594,E2 19509.594} C_VEL
LIN {X 0,Y 401.477,Z 376.788,A -85,B 0,C 180,E1 19505.715,E2 19505.715} C_VEL
LIN {X 0,Y 401.478,Z 376.79,A -85,B 0,C 180,E1 19501.759,E2 19501.759} C_VEL
LIN {X 0,Y 401.467,Z 376.792,A -85,B 0,C 180,E1 19497.863,E2 19497.863} C_VEL
LIN {X 0,Y 401.452,Z 376.795,A -85,B 0,C 180,E1 19494,E2 19494} C_VEL
LIN {X 0,Y 401.438,Z 376.794,A -85,B 0,C 180,E1 19490.2,E2 19490.2} C_VEL
LIN {X 0,Y 401.431,Z 376.792,A -85,B 0,C 180,E1 19486.375,E2 19486.375} C_VEL
LIN {X 0,Y 401.43,Z 376.794,A -85,B 0,C 180,E1 19482.454,E2 19482.454} C_VEL
LIN {X 0,Y 401.431,Z 376.795,A -85,B 0,C 180,E1 19478.513,E2 19478.513} C_VEL
LIN {X 0,Y 401.453,Z 376.949,A -85,B 0,C 180,E1 19476.582,E2 19476.582} C_VEL
LIN {X 0,Y 406.877,Z 396.327,A -85,B 0,C 180,E1 19472.978,E2 19472.978} C_VEL
LIN {X 0,Y 410.74,Z 411.491,A -85,B 0,C 180,E1 19470.299,E2 19470.299} C_VEL
LIN {X 0,Y 408.479,Z 438.087,A -85,B 0,C 180,E1 19466.377,E2 19466.377} C_VEL
LIN {X 0,Y 406.268,Z 466.863,A -85,B 0,C 180,E1 19462.196,E2 19462.196} C_VEL
LIN {X 0,Y 405.512,Z 478.934,A -85,B 0,C 180,E1 19460.505,E2 19460.505} C_VEL
LIN {X 0,Y 408.893,Z 504.442,A -85,B 0,C 180,E1 19459.702,E2 19459.702} C_VEL
LIN {X 0,Y 406.216,Z 603.683,A -85,B 0,C 180,E1 19457.397,E2 19457.397} C_VEL
LIN {X 0,Y 405.753,Z 619.831,A -85,B 0,C 180,E1 19456.757,E2 19456.757} C_VEL
LIN {X 0,Y 405.159,Z 634.999,A -85,B 0,C 180,E1 19455.898,E2 19455.898} C_VEL
LIN {X 0,Y 404.346,Z 650.869,A -85,B 0,C 180,E1 19454.683,E2 19454.683} C_VEL
LIN {X 0,Y 403.581,Z 665.113,A -85,B 0,C 180,E1 19453.248,E2 19453.248} C_VEL
LIN {X 0,Y 402.854,Z 677.869,A -85,B 0,C 180,E1 19451.598,E2 19451.598} C_VEL
LIN {X 0,Y 402.263,Z 688.325,A -85,B 0,C 180,E1 19449.876,E2 19449.876} C_VEL
LIN {X 0,Y 401.842,Z 696.646,A -85,B 0,C 180,E1 19448.154,E2 19448.154} C_VEL
LIN {X 0,Y 401.526,Z 704.071,A -85,B 0,C 180,E1 19446.147,E2 19446.147} C_VEL
LIN {X 0,Y 401.355,Z 709.447,A -85,B 0,C 180,E1 19444.143,E2 19444.143} C_VEL
LIN {X 0,Y 401.33,Z 713.037,A -85,B 0,C 180,E1 19442.142,E2 19442.142} C_VEL
LIN {X 0,Y 401.401,Z 714.948,A -85,B 0,C 180,E1 19440,E2 19440} C_VEL
LIN {X 0,Y 401.599,Z 715.064,A -85,B 0,C 180,E1 19438.003,E2 19438.003} C_VEL
LIN {X 0,Y 401.907,Z 713.271,A -85,B 0,C 180,E1 19435.863,E2 19435.863} C_VEL
LIN {X 0,Y 402.358,Z 709.808,A -85,B 0,C 180,E1 19433.866,E2 19433.866} C_VEL
LIN {X 0,Y 402.985,Z 704.496,A -85,B 0,C 180,E1 19431.87,E2 19431.87} C_VEL
LIN {X 0,Y 403.731,Z 697.661,A -85,B 0,C 180,E1 19430.017,E2 19430.017} C_VEL
LIN {X 0,Y 404.69,Z 688.686,A -85,B 0,C 180,E1 19428.167,E2 19428.167} C_VEL
LIN {X 0,Y 405.765,Z 678.015,A -85,B 0,C 180,E1 19426.462,E2 19426.462} C_VEL
LIN {X 0,Y 406.848,Z 666.305,A -85,B 0,C 180,E1 19424.98,E2 19424.98} C_VEL
LIN {X 0,Y 407.93,Z 653.618,A -85,B 0,C 180,E1 19423.701,E2 19423.701} C_VEL
LIN {X 0,Y 409.096,Z 638.375,A -85,B 0,C 180,E1 19422.505,E2 19422.505} C_VEL
LIN {X 0,Y 410.147,Z 621.696,A -85,B 0,C 180,E1 19421.524,E2 19421.524} C_VEL
LIN {X 0,Y 411.014,Z 603.982,A -85,B 0,C 180,E1 19420.8,E2 19420.8} C_VEL
LIN {X 0,Y 417.386,Z 514.111,A -85,B 0,C 180,E1 19417.954,E2 19417.954} C_VEL
LIN {X 0,Y 417.734,Z 507.551,A -85,B 0,C 180,E1 19417.724,E2 19417.724} C_VEL
LIN {X 0,Y 414.719,Z 488.026,A -85,B 0,C 180,E1 19416.544,E2 19416.544} C_VEL
LIN {X 0,Y 412.942,Z 478.339,A -85,B 0,C 180,E1 19415.845,E2 19415.845} C_VEL
LIN {X 0,Y 417.239,Z 453.238,A -85,B 0,C 180,E1 19411.675,E2 19411.675} C_VEL
LIN {X 0,Y 422.217,Z 431.477,A -85,B 0,C 180,E1 19407.804,E2 19407.804} C_VEL
LIN {X 0,Y 421.324,Z 424.482,A -85,B 0,C 180,E1 19405.776,E2 19405.776} C_VEL
LIN {X 0,Y 420.186,Z 418.444,A -85,B 0,C 180,E1 19403.495,E2 19403.495} C_VEL
LIN {X 0,Y 419.293,Z 414.612,A -85,B 0,C 180,E1 19401.459,E2 19401.459} C_VEL
LIN {X 0,Y 418.876,Z 412.76,A -85,B 0,C 180,E1 19400.017,E2 19400.017} C_VEL
LIN {X 0,Y 418.926,Z 411.085,A -85,B 0,C 180,E1 19397.512,E2 19397.512} C_VEL
LIN {X 0,Y 419.17,Z 411.363,A -85,B 0,C 180,E1 19396.042,E2 19396.042} C_VEL
LIN {X 0,Y 420.071,Z 414.115,A -85,B 0,C 180,E1 19393.451,E2 19393.451} C_VEL
LIN {X 0,Y 420.911,Z 416.466,A -85,B 0,C 180,E1 19392.171,E2 19392.171} C_VEL
LIN {X 0,Y 422.439,Z 420.631,A -85,B 0,C 180,E1 19390.431,E2 19390.431} C_VEL
LIN {X 0,Y 424.282,Z 427.201,A -85,B 0,C 180,E1 19388.473,E2 19388.473} C_VEL
LIN {X 0,Y 425.391,Z 432.454,A -85,B 0,C 180,E1 19387.246,E2 19387.246} C_VEL
LIN {X 0,Y 419.866,Z 455.575,A -85,B 0,C 180,E1 19384.36,E2 19384.36} C_VEL
LIN {X 0,Y 417.518,Z 469.04,A -85,B 0,C 180,E1 19382.816,E2 19382.816} C_VEL
LIN {X 0,Y 419.293,Z 490.155,A -85,B 0,C 180,E1 19381.974,E2 19381.974} C_VEL
LIN {X 0,Y 417.499,Z 532.593,A -85,B 0,C 180,E1 19381.008,E2 19381.008} C_VEL
LIN {X 0,Y 413.171,Z 668.027,A -85,B 0,C 180,E1 19378.123,E2 19378.123} C_VEL
LIN {X 0,Y 412.028,Z 687.505,A -85,B 0,C 180,E1 19377.456,E2 19377.456} C_VEL
LIN {X 0,Y 410.58,Z 706.816,A -85,B 0,C 180,E1 19376.52,E2 19376.52} C_VEL
LIN {X 0,Y 409.055,Z 724.339,A -85,B 0,C 180,E1 19375.403,E2 19375.403} C_VEL
LIN {X 0,Y 407.441,Z 741.36,A -85,B 0,C 180,E1 19374.04,E2 19374.04} C_VEL
LIN {X 0,Y 405.823,Z 757.478,A -85,B 0,C 180,E1 19372.451,E2 19372.451} C_VEL
LIN {X 0,Y 404.287,Z 772.596,A -85,B 0,C 180,E1 19370.636,E2 19370.636} C_VEL
LIN {X 0,Y 402.958,Z 786.108,A -85,B 0,C 180,E1 19368.668,E2 19368.668} C_VEL
LIN {X 0,Y 401.821,Z 798.52,A -85,B 0,C 180,E1 19366.479,E2 19366.479} C_VEL
LIN {X 0,Y 401.048,Z 808.753,A -85,B 0,C 180,E1 19364.289,E2 19364.289} C_VEL
LIN {X 0,Y 400.507,Z 817.605,A -85,B 0,C 180,E1 19361.959,E2 19361.959} C_VEL
LIN {X 0,Y 400.234,Z 824.998,A -85,B 0,C 180,E1 19359.49,E2 19359.49} C_VEL
LIN {X 0,Y 400.169,Z 830.542,A -85,B 0,C 180,E1 19357.032,E2 19357.032} C_VEL
LIN {X 0,Y 400.178,Z 834.464,A -85,B 0,C 180,E1 19354.503,E2 19354.503} C_VEL
LIN {X 0,Y 400.233,Z 836.629,A -85,B 0,C 180,E1 19352.004,E2 19352.004} C_VEL
LIN {X 0,Y 400.251,Z 837.135,A -85,B 0,C 180,E1 19349.571,E2 19349.571} C_VEL
LIN {X 0,Y 400.216,Z 836.056,A -85,B 0,C 180,E1 19347.136,E2 19347.136} C_VEL
LIN {X 0,Y 400.165,Z 833.152,A -85,B 0,C 180,E1 19344.552,E2 19344.552} C_VEL
LIN {X 0,Y 400.168,Z 828.725,A -85,B 0,C 180,E1 19342.101,E2 19342.101} C_VEL
LIN {X 0,Y 400.301,Z 822.534,A -85,B 0,C 180,E1 19339.64,E2 19339.64} C_VEL
LIN {X 0,Y 400.679,Z 814.437,A -85,B 0,C 180,E1 19337.168,E2 19337.168} C_VEL
LIN {X 0,Y 401.315,Z 804.866,A -85,B 0,C 180,E1 19334.835,E2 19334.835} C_VEL
LIN {X 0,Y 402.241,Z 793.909,A -85,B 0,C 180,E1 19332.645,E2 19332.645} C_VEL
LIN {X 0,Y 403.482,Z 781.128,A -85,B 0,C 180,E1 19330.531,E2 19330.531} C_VEL
LIN {X 0,Y 404.992,Z 766.728,A -85,B 0,C 180,E1 19328.552,E2 19328.552} C_VEL
LIN {X 0,Y 406.714,Z 750.992,A -85,B 0,C 180,E1 19326.761,E2 19326.761} C_VEL
LIN {X 0,Y 408.54,Z 734.161,A -85,B 0,C 180,E1 19325.182,E2 19325.182} C_VEL
LIN {X 0,Y 410.398,Z 716.486,A -85,B 0,C 180,E1 19323.834,E2 19323.834} C_VEL
LIN {X 0,Y 412.224,Z 698.062,A -85,B 0,C 180,E1 19322.714,E2 19322.714} C_VEL
LIN {X 0,Y 413.995,Z 678.014,A -85,B 0,C 180,E1 19321.79,E2 19321.79} C_VEL
LIN {X 0,Y 415.431,Z 657.549,A -85,B 0,C 180,E1 19321.122,E2 19321.122} C_VEL
LIN {X 0,Y 420.19,Z 570.02,A -85,B 0,C 180,E1 19318.892,E2 19318.892} C_VEL
LIN {X 0,Y 426.036,Z 490.112,A -85,B 0,C 180,E1 19316.679,E2 19316.679} C_VEL
LIN {X 0,Y 424.993,Z 463.253,A -85,B 0,C 180,E1 19315.362,E2 19315.362} C_VEL
LIN {X 0,Y 423.899,Z 440.369,A -85,B 0,C 180,E1 19314.044,E2 19314.044} C_VEL
LIN {X 0,Y 423.819,Z 427.325,A -85,B 0,C 180,E1 19313.124,E2 19313.124} C_VEL
LIN {X 0,Y 420.956,Z 416.146,A -85,B 0,C 180,E1 19311.423,E2 19311.423} C_VEL
LIN {X 0,Y 419.312,Z 405.341,A -85,B 0,C 180,E1 19309.523,E2 19309.523} C_VEL
LIN {X 0,Y 418.803,Z 400.868,A -85,B 0,C 180,E1 19308.457,E2 19308.457} C_VEL
LIN {X 0,Y 417.084,Z 398.836,A -85,B 0,C 180,E1 19306.337,E2 19306.337} C_VEL
LIN {X 0,Y 416.717,Z 398.702,A -85,B 0,C 180,E1 19304.863,E2 19304.863} C_VEL
LIN {X 0,Y 417.503,Z 400.423,A -85,B 0,C 180,E1 19302.471,E2 19302.471} C_VEL
LIN {X 0,Y 418.041,Z 401.1,A -85,B 0,C 180,E1 19301.859,E2 19301.859} C_VEL
LIN {X 0,Y 419.36,Z 404.667,A -85,B 0,C 180,E1 19300.25,E2 19300.25} C_VEL
LIN {X 0,Y 421.401,Z 409.986,A -85,B 0,C 180,E1 19298.464,E2 19298.464} C_VEL
LIN {X 0,Y 423.369,Z 415.387,A -85,B 0,C 180,E1 19297.029,E2 19297.029} C_VEL
LIN {X 0,Y 425.369,Z 421.884,A -85,B 0,C 180,E1 19295.632,E2 19295.632} C_VEL
LIN {X 0,Y 429.061,Z 430.243,A -85,B 0,C 180,E1 19294.482,E2 19294.482} C_VEL
LIN {X 0,Y 429.634,Z 432.59,A -85,B 0,C 180,E1 19294.266,E2 19294.266} C_VEL
LIN {X 0,Y 430.147,Z 439.791,A -85,B 0,C 180,E1 19293.848,E2 19293.848} C_VEL
LIN {X 0,Y 422.709,Z 526.799,A -85,B 0,C 180,E1 19291.422,E2 19291.422} C_VEL
LIN {X 0,Y 418.054,Z 600.844,A -85,B 0,C 180,E1 19289.491,E2 19289.491} C_VEL
LIN {X 0,Y 416.596,Z 629.615,A -85,B 0,C 180,E1 19288.711,E2 19288.711} C_VEL
LIN {X 0,Y 415.288,Z 649.148,A -85,B 0,C 180,E1 19287.92,E2 19287.92} C_VEL
LIN {X 0,Y 413.702,Z 668.328,A -85,B 0,C 180,E1 19286.869,E2 19286.869} C_VEL
LIN {X 0,Y 411.941,Z 686.395,A -85,B 0,C 180,E1 19285.597,E2 19285.597} C_VEL
LIN {X 0,Y 410.064,Z 703.296,A -85,B 0,C 180,E1 19284.105,E2 19284.105} C_VEL
LIN {X 0,Y 408.238,Z 718.51,A -85,B 0,C 180,E1 19282.462,E2 19282.462} C_VEL
LIN {X 0,Y 406.435,Z 732.77,A -85,B 0,C 180,E1 19280.597,E2 19280.597} C_VEL
LIN {X 0,Y 404.803,Z 745.518,A -85,B 0,C 180,E1 19278.58,E2 19278.58} C_VEL
LIN {X 0,Y 403.387,Z 756.813,A -85,B 0,C 180,E1 19276.413,E2 19276.413} C_VEL
LIN {X 0,Y 402.222,Z 766.655,A -85,B 0,C 180,E1 19274.1,E2 19274.1} C_VEL
LIN {X 0,Y 401.33,Z 775.007,A -85,B 0,C 180,E1 19271.642,E2 19271.642} C_VEL
LIN {X 0,Y 400.719,Z 781.8,A -85,B 0,C 180,E1 19269.044,E2 19269.044} C_VEL
LIN {X 0,Y 400.361,Z 786.656,A -85,B 0,C 180,E1 19266.453,E2 19266.453} C_VEL
LIN {X 0,Y 400.182,Z 789.741,A -85,B 0,C 180,E1 19263.868,E2 19263.868} C_VEL
LIN {X 0,Y 400.108,Z 791.14,A -85,B 0,C 180,E1 19261.289,E2 19261.289} C_VEL
LIN {X 0,Y 400.085,Z 790.875,A -85,B 0,C 180,E1 19258.711,E2 19258.711} C_VEL
LIN {X 0,Y 400.116,Z 788.942,A -85,B 0,C 180,E1 19256.131,E2 19256.131} C_VEL
LIN {X 0,Y 400.238,Z 785.298,A -85,B 0,C 180,E1 19253.545,E2 19253.545} C_VEL
LIN {X 0,Y 400.492,Z 780.209,A -85,B 0,C 180,E1 19251.095,E2 19251.095} C_VEL
LIN {X 0,Y 400.95,Z 773.374,A -85,B 0,C 180,E1 19248.638,E2 19248.638} C_VEL
LIN {X 0,Y 401.626,Z 765.176,A -85,B 0,C 180,E1 19246.319,E2 19246.319} C_VEL
LIN {X 0,Y 402.604,Z 754.85,A -85,B 0,C 180,E1 19243.969,E2 19243.969} C_VEL
LIN {X 0,Y 403.799,Z 743.325,A -85,B 0,C 180,E1 19241.82,E2 19241.82} C_VEL
LIN {X 0,Y 405.277,Z 729.647,A -85,B 0,C 180,E1 19239.719,E2 19239.719} C_VEL
LIN {X 0,Y 406.881,Z 714.806,A -85,B 0,C 180,E1 19237.839,E2 19237.839} C_VEL
LIN {X 0,Y 408.522,Z 698.906,A -85,B 0,C 180,E1 19236.181,E2 19236.181} C_VEL
LIN {X 0,Y 410.138,Z 681.977,A -85,B 0,C 180,E1 19234.746,E2 19234.746} C_VEL
LIN {X 0,Y 411.653,Z 663.985,A -85,B 0,C 180,E1 19233.532,E2 19233.532} C_VEL
LIN {X 0,Y 412.949,Z 645.224,A -85,B 0,C 180,E1 19232.552,E2 19232.552} C_VEL
LIN {X 0,Y 414.034,Z 625.142,A -85,B 0,C 180,E1 19231.793,E2 19231.793} C_VEL
LIN {X 0,Y 414.821,Z 602.775,A -85,B 0,C 180,E1 19231.248,E2 19231.248} C_VEL
LIN {X 0,Y 420.31,Z 434.907,A -85,B 0,C 180,E1 19227.724,E2 19227.724} C_VEL
LIN {X 0,Y 417.656,Z 420.367,A -85,B 0,C 180,E1 19227.171,E2 19227.171} C_VEL
LIN {X 0,Y 412.857,Z 409.97,A -85,B 0,C 180,E1 19226.532,E2 19226.532} C_VEL
LIN {X 0,Y 405.46,Z 388.201,A -85,B 0,C 180,E1 19223.506,E2 19223.506} C_VEL
LIN {X 0,Y 401.442,Z 376.791,A -85,B 0,C 180,E1 19221.852,E2 19221.852} C_VEL
LIN {X 0,Y 401.462,Z 376.793,A -85,B 0,C 180,E1 19218.128,E2 19218.128} C_VEL
LIN {X 0,Y 401.472,Z 376.791,A -85,B 0,C 180,E1 19214.214,E2 19214.214} C_VEL
LIN {X 0,Y 401.49,Z 376.788,A -85,B 0,C 180,E1 19210.353,E2 19210.353} C_VEL
LIN {X 0,Y 401.479,Z 376.79,A -85,B 0,C 180,E1 19206.351,E2 19206.351} C_VEL
LIN {X 0,Y 401.479,Z 376.791,A -85,B 0,C 180,E1 19202.374,E2 19202.374} C_VEL
LIN {X 0,Y 401.48,Z 376.789,A -85,B 0,C 180,E1 19198.403,E2 19198.403} C_VEL
LIN {X 0,Y 401.473,Z 376.79,A -85,B 0,C 180,E1 19194.42,E2 19194.42} C_VEL
LIN {X 0,Y 401.458,Z 376.788,A -85,B 0,C 180,E1 19190.559,E2 19190.559} C_VEL
LIN {X 0,Y 401.442,Z 376.786,A -85,B 0,C 180,E1 19186.793,E2 19186.793} C_VEL
LIN {X 0,Y 401.445,Z 376.792,A -85,B 0,C 180,E1 19184.658,E2 19184.658} C_VEL
LIN {X 0,Y 400.517,Z 376.914,A -85,B 0,C 180,E1 19183.558,E2 19183.558} C_VEL
LIN {X 0,Y 395.953,Z 377.484,A -85,B 0,C 180,E1 19181.484,E2 19181.484} C_VEL
LIN {X 0,Y 393.684,Z 377.76,A -85,B 0,C 180,E1 19180.055,E2 19180.055} C_VEL
LIN {X 0,Y 393.515,Z 377.776,A -85,B 0,C 180,E1 19179.648,E2 19179.648} C_VEL
LIN {X 0,Y 393.532,Z 377.778,A -85,B 0,C 180,E1 19175.833,E2 19175.833} C_VEL
LIN {X 0,Y 393.535,Z 377.778,A -85,B 0,C 180,E1 19171.893,E2 19171.893} C_VEL
LIN {X 0,Y 393.537,Z 377.771,A -85,B 0,C 180,E1 19167.962,E2 19167.962} C_VEL
LIN {X 0,Y 393.543,Z 377.777,A -85,B 0,C 180,E1 19163.874,E2 19163.874} C_VEL
LIN {X 0,Y 393.537,Z 377.779,A -85,B 0,C 180,E1 19159.903,E2 19159.903} C_VEL
LIN {X 0,Y 393.544,Z 377.778,A -85,B 0,C 180,E1 19155.883,E2 19155.883} C_VEL
LIN {X 0,Y 393.537,Z 377.779,A -85,B 0,C 180,E1 19151.79,E2 19151.79} C_VEL
LIN {X 0,Y 393.55,Z 377.778,A -85,B 0,C 180,E1 19147.756,E2 19147.756} C_VEL
LIN {X 0,Y 393.537,Z 377.779,A -85,B 0,C 180,E1 19143.75,E2 19143.75} C_VEL
LIN {X 0,Y 393.54,Z 377.778,A -85,B 0,C 180,E1 19139.75,E2 19139.75} C_VEL
LIN {X 0,Y 393.535,Z 377.782,A -85,B 0,C 180,E1 19135.663,E2 19135.663} C_VEL
LIN {X 0,Y 393.535,Z 377.781,A -85,B 0,C 180,E1 19131.688,E2 19131.688} C_VEL
LIN {X 0,Y 393.532,Z 377.78,A -85,B 0,C 180,E1 19127.677,E2 19127.677} C_VEL
LIN {X 0,Y 393.531,Z 377.78,A -85,B 0,C 180,E1 19123.605,E2 19123.605} C_VEL
LIN {X 0,Y 393.528,Z 377.782,A -85,B 0,C 180,E1 19119.659,E2 19119.659} C_VEL
LIN {X 0,Y 393.533,Z 377.832,A -85,B 0,C 180,E1 19117.157,E2 19117.157} C_VEL
LIN {X 0,Y 398.988,Z 397.424,A -85,B 0,C 180,E1 19113.436,E2 19113.436} C_VEL
LIN {X 0,Y 403.118,Z 413.902,A -85,B 0,C 180,E1 19110.479,E2 19110.479} C_VEL
LIN {X 0,Y 400.762,Z 440.324,A -85,B 0,C 180,E1 19106.525,E2 19106.525} C_VEL
LIN {X 0,Y 398.486,Z 468.678,A -85,B 0,C 180,E1 19102.342,E2 19102.342} C_VEL
LIN {X 0,Y 397.829,Z 478.814,A -85,B 0,C 180,E1 19100.907,E2 19100.907} C_VEL
LIN {X 0,Y 401.298,Z 505.333,A -85,B 0,C 180,E1 19100.049,E2 19100.049} C_VEL
LIN {X 0,Y 398.487,Z 604.19,A -85,B 0,C 180,E1 19097.684,E2 19097.684} C_VEL
LIN {X 0,Y 398.022,Z 619.894,A -85,B 0,C 180,E1 19097.055,E2 19097.055} C_VEL
LIN {X 0,Y 397.377,Z 635.762,A -85,B 0,C 180,E1 19096.143,E2 19096.143} C_VEL
LIN {X 0,Y 396.533,Z 651.66,A -85,B 0,C 180,E1 19094.904,E2 19094.904} C_VEL
LIN {X 0,Y 395.739,Z 665.96,A -85,B 0,C 180,E1 19093.441,E2 19093.441} C_VEL
LIN {X 0,Y 394.983,Z 678.771,A -85,B 0,C 180,E1 19091.758,E2 19091.758} C_VEL
LIN {X 0,Y 394.39,Z 688.888,A -85,B 0,C 180,E1 19090.075,E2 19090.075} C_VEL
LIN {X 0,Y 393.945,Z 697.348,A -85,B 0,C 180,E1 19088.318,E2 19088.318} C_VEL
LIN {X 0,Y 393.609,Z 704.892,A -85,B 0,C 180,E1 19086.271,E2 19086.271} C_VEL
LIN {X 0,Y 393.443,Z 710.095,A -85,B 0,C 180,E1 19084.373,E2 19084.373} C_VEL
LIN {X 0,Y 393.41,Z 714.126,A -85,B 0,C 180,E1 19082.185,E2 19082.185} C_VEL
LIN {X 0,Y 393.485,Z 716.089,A -85,B 0,C 180,E1 19080.146,E2 19080.146} C_VEL
LIN {X 0,Y 393.714,Z 716.387,A -85,B 0,C 180,E1 19077.963,E2 19077.963} C_VEL
LIN {X 0,Y 394.057,Z 714.706,A -85,B 0,C 180,E1 19075.78,E2 19075.78} C_VEL
LIN {X 0,Y 394.562,Z 711.392,A -85,B 0,C 180,E1 19073.744,E2 19073.744} C_VEL
LIN {X 0,Y 395.298,Z 705.726,A -85,B 0,C 180,E1 19071.564,E2 19071.564} C_VEL
LIN {X 0,Y 396.122,Z 698.845,A -85,B 0,C 180,E1 19069.676,E2 19069.676} C_VEL
LIN {X 0,Y 397.187,Z 689.901,A -85,B 0,C 180,E1 19067.792,E2 19067.792} C_VEL
LIN {X 0,Y 398.408,Z 678.794,A -85,B 0,C 180,E1 19065.993,E2 19065.993} C_VEL
LIN {X 0,Y 399.719,Z 665.582,A -85,B 0,C 180,E1 19064.327,E2 19064.327} C_VEL
LIN {X 0,Y 401,Z 651.721,A -85,B 0,C 180,E1 19062.964,E2 19062.964} C_VEL
LIN {X 0,Y 402.122,Z 637.794,A -85,B 0,C 180,E1 19061.892,E2 19061.892} C_VEL
LIN {X 0,Y 403.226,Z 621.425,A -85,B 0,C 180,E1 19060.932,E2 19060.932} C_VEL
LIN {X 0,Y 404.19,Z 603.712,A -85,B 0,C 180,E1 19060.2,E2 19060.2} C_VEL
LIN {X 0,Y 411.376,Z 511.749,A -85,B 0,C 180,E1 19057.176,E2 19057.176} C_VEL
LIN {X 0,Y 411.269,Z 507.881,A -85,B 0,C 180,E1 19056.995,E2 19056.995} C_VEL
LIN {X 0,Y 408.349,Z 488.42,A -85,B 0,C 180,E1 19055.737,E2 19055.737} C_VEL
LIN {X 0,Y 406.468,Z 478.3,A -85,B 0,C 180,E1 19054.97,E2 19054.97} C_VEL
LIN {X 0,Y 411.223,Z 453.688,A -85,B 0,C 180,E1 19050.744,E2 19050.744} C_VEL
LIN {X 0,Y 415.973,Z 435.205,A -85,B 0,C 180,E1 19047.342,E2 19047.342} C_VEL
LIN {X 0,Y 415.075,Z 428.487,A -85,B 0,C 180,E1 19045.228,E2 19045.228} C_VEL
LIN {X 0,Y 414.215,Z 423.178,A -85,B 0,C 180,E1 19043.034,E2 19043.034} C_VEL
LIN {X 0,Y 413.592,Z 419.199,A -85,B 0,C 180,E1 19040.679,E2 19040.679} C_VEL
LIN {X 0,Y 413.419,Z 417.106,A -85,B 0,C 180,E1 19037.939,E2 19037.939} C_VEL
LIN {X 0,Y 413.736,Z 417.12,A -85,B 0,C 180,E1 19036.268,E2 19036.268} C_VEL
LIN {X 0,Y 414.518,Z 419.786,A -85,B 0,C 180,E1 19033.645,E2 19033.645} C_VEL
LIN {X 0,Y 415.174,Z 421.648,A -85,B 0,C 180,E1 19032.529,E2 19032.529} C_VEL
LIN {X 0,Y 416.556,Z 425.701,A -85,B 0,C 180,E1 19030.76,E2 19030.76} C_VEL
LIN {X 0,Y 418.278,Z 432.002,A -85,B 0,C 180,E1 19028.777,E2 19028.777} C_VEL
LIN {X 0,Y 419.116,Z 436.235,A -85,B 0,C 180,E1 19027.728,E2 19027.728} C_VEL
LIN {X 0,Y 413.26,Z 458.877,A -85,B 0,C 180,E1 19024.819,E2 19024.819} C_VEL
LIN {X 0,Y 411.271,Z 469.41,A -85,B 0,C 180,E1 19023.579,E2 19023.579} C_VEL
LIN {X 0,Y 412.775,Z 486.718,A -85,B 0,C 180,E1 19022.815,E2 19022.815} C_VEL
LIN {X 0,Y 412.885,Z 493.371,A -85,B 0,C 180,E1 19022.589,E2 19022.589} C_VEL
LIN {X 0,Y 408.484,Z 585.933,A -85,B 0,C 180,E1 19020.352,E2 19020.352} C_VEL
LIN {X 0,Y 405.758,Z 667.7,A -85,B 0,C 180,E1 19018.548,E2 19018.548} C_VEL
LIN {X 0,Y 404.575,Z 686.992,A -85,B 0,C 180,E1 19017.876,E2 19017.876} C_VEL
LIN {X 0,Y 403.161,Z 705.118,A -85,B 0,C 180,E1 19016.991,E2 19016.991} C_VEL
LIN {X 0,Y 401.537,Z 723.198,A -85,B 0,C 180,E1 19015.834,E2 19015.834} C_VEL
LIN {X 0,Y 399.863,Z 740.109,A -85,B 0,C 180,E1 19014.47,E2 19014.47} C_VEL
LIN {X 0,Y 398.208,Z 755.903,A -85,B 0,C 180,E1 19012.904,E2 19012.904} C_VEL
LIN {X 0,Y 396.578,Z 771.249,A -85,B 0,C 180,E1 19011.056,E2 19011.056} C_VEL
LIN {X 0,Y 395.169,Z 784.98,A -85,B 0,C 180,E1 19009.05,E2 19009.05} C_VEL
LIN {X 0,Y 393.96,Z 797.531,A -85,B 0,C 180,E1 19006.818,E2 19006.818} C_VEL
LIN {X 0,Y 393.084,Z 808.479,A -85,B 0,C 180,E1 19004.435,E2 19004.435} C_VEL
LIN {X 0,Y 392.512,Z 817.525,A -85,B 0,C 180,E1 19001.992,E2 19001.992} C_VEL
LIN {X 0,Y 392.233,Z 824.985,A -85,B 0,C 180,E1 18999.419,E2 18999.419} C_VEL
LIN {X 0,Y 392.171,Z 830.466,A -85,B 0,C 180,E1 18996.882,E2 18996.882} C_VEL
LIN {X 0,Y 392.195,Z 834.312,A -85,B 0,C 180,E1 18994.24,E2 18994.24} C_VEL
LIN {X 0,Y 392.256,Z 836.32,A -85,B 0,C 180,E1 18991.607,E2 18991.607} C_VEL
LIN {X 0,Y 392.27,Z 836.564,A -85,B 0,C 180,E1 18989.124,E2 18989.124} C_VEL
LIN {X 0,Y 392.212,Z 835.079,A -85,B 0,C 180,E1 18986.492,E2 18986.492} C_VEL
LIN {X 0,Y 392.167,Z 831.786,A -85,B 0,C 180,E1 18983.853,E2 18983.853} C_VEL
LIN {X 0,Y 392.192,Z 826.621,A -85,B 0,C 180,E1 18981.201,E2 18981.201} C_VEL
LIN {X 0,Y 392.41,Z 819.894,A -85,B 0,C 180,E1 18978.685,E2 18978.685} C_VEL
LIN {X 0,Y 392.924,Z 811.219,A -85,B 0,C 180,E1 18976.161,E2 18976.161} C_VEL
LIN {X 0,Y 393.732,Z 801.033,A -85,B 0,C 180,E1 18973.779,E2 18973.779} C_VEL
LIN {X 0,Y 394.874,Z 789.408,A -85,B 0,C 180,E1 18971.548,E2 18971.548} C_VEL
LIN {X 0,Y 396.411,Z 775.381,A -85,B 0,C 180,E1 18969.322,E2 18969.322} C_VEL
LIN {X 0,Y 398.192,Z 760.077,A -85,B 0,C 180,E1 18967.329,E2 18967.329} C_VEL
LIN {X 0,Y 400.127,Z 743.711,A -85,B 0,C 180,E1 18965.571,E2 18965.571} C_VEL
LIN {X 0,Y 402.136,Z 726.409,A -85,B 0,C 180,E1 18964.049,E2 18964.049} C_VEL
LIN {X 0,Y 404.279,Z 707.211,A -85,B 0,C 180,E1 18962.692,E2 18962.692} C_VEL
LIN {X 0,Y 406.32,Z 687.393,A -85,B 0,C 180,E1 18961.605,E2 18961.605} C_VEL
LIN {X 0,Y 408.125,Z 666.905,A -85,B 0,C 180,E1 18960.786,E2 18960.786} C_VEL
LIN {X 0,Y 409.971,Z 636.02,A -85,B 0,C 180,E1 18959.937,E2 18959.937} C_VEL
LIN {X 0,Y 414.981,Z 558.632,A -85,B 0,C 180,E1 18957.852,E2 18957.852} C_VEL
LIN {X 0,Y 420.556,Z 491.285,A -85,B 0,C 180,E1 18955.9,E2 18955.9} C_VEL
LIN {X 0,Y 419.866,Z 463.742,A -85,B 0,C 180,E1 18954.481,E2 18954.481} C_VEL
LIN {X 0,Y 419.19,Z 440.793,A -85,B 0,C 180,E1 18953.085,E2 18953.085} C_VEL
LIN {X 0,Y 419.252,Z 431.556,A -85,B 0,C 180,E1 18952.402,E2 18952.402} C_VEL
LIN {X 0,Y 416.563,Z 418.672,A -85,B 0,C 180,E1 18950.322,E2 18950.322} C_VEL
LIN {X 0,Y 415.778,Z 410.583,A -85,B 0,C 180,E1 18948.783,E2 18948.783} C_VEL
LIN {X 0,Y 415.644,Z 408.117,A -85,B 0,C 180,E1 18948.214,E2 18948.214} C_VEL
LIN {X 0,Y 414.019,Z 406.156,A -85,B 0,C 180,E1 18946.123,E2 18946.123} C_VEL
LIN {X 0,Y 413.586,Z 406.231,A -85,B 0,C 180,E1 18944.506,E2 18944.506} C_VEL
LIN {X 0,Y 414.491,Z 408.285,A -85,B 0,C 180,E1 18942.014,E2 18942.014} C_VEL
LIN {X 0,Y 415.891,Z 412.677,A -85,B 0,C 180,E1 18940.029,E2 18940.029} C_VEL
LIN {X 0,Y 417.493,Z 417.449,A -85,B 0,C 180,E1 18938.451,E2 18938.451} C_VEL
LIN {X 0,Y 419.268,Z 423.126,A -85,B 0,C 180,E1 18936.974,E2 18936.974} C_VEL
LIN {X 0,Y 423.029,Z 431.262,A -85,B 0,C 180,E1 18935.603,E2 18935.603} C_VEL
LIN {X 0,Y 424.824,Z 436.459,A -85,B 0,C 180,E1 18934.957,E2 18934.957} C_VEL
LIN {X 0,Y 425.058,Z 441.816,A -85,B 0,C 180,E1 18934.647,E2 18934.647} C_VEL
LIN {X 0,Y 416.893,Z 527.573,A -85,B 0,C 180,E1 18932.164,E2 18932.164} C_VEL
LIN {X 0,Y 411.451,Z 605.138,A -85,B 0,C 180,E1 18930.054,E2 18930.054} C_VEL
LIN {X 0,Y 410.003,Z 630.752,A -85,B 0,C 180,E1 18929.322,E2 18929.322} C_VEL
LIN {X 0,Y 408.569,Z 650.272,A -85,B 0,C 180,E1 18928.503,E2 18928.503} C_VEL
LIN {X 0,Y 406.863,Z 669.195,A -85,B 0,C 180,E1 18927.437,E2 18927.437} C_VEL
LIN {X 0,Y 404.976,Z 687.084,A -85,B 0,C 180,E1 18926.149,E2 18926.149} C_VEL
LIN {X 0,Y 402.962,Z 703.885,A -85,B 0,C 180,E1 18924.636,E2 18924.636} C_VEL
LIN {X 0,Y 400.92,Z 719.628,A -85,B 0,C 180,E1 18922.895,E2 18922.895} C_VEL
LIN {X 0,Y 398.922,Z 734.257,A -85,B 0,C 180,E1 18920.926,E2 18920.926} C_VEL
LIN {X 0,Y 397.123,Z 747.281,A -85,B 0,C 180,E1 18918.794,E2 18918.794} C_VEL
LIN {X 0,Y 395.625,Z 758.328,A -85,B 0,C 180,E1 18916.594,E2 18916.594} C_VEL
LIN {X 0,Y 394.387,Z 767.984,A -85,B 0,C 180,E1 18914.236,E2 18914.236} C_VEL
LIN {X 0,Y 393.436,Z 776.166,A -85,B 0,C 180,E1 18911.73,E2 18911.73} C_VEL
LIN {X 0,Y 392.777,Z 782.759,A -85,B 0,C 180,E1 18909.081,E2 18909.081} C_VEL
LIN {X 0,Y 392.393,Z 787.458,A -85,B 0,C 180,E1 18906.437,E2 18906.437} C_VEL
LIN {X 0,Y 392.201,Z 790.4,A -85,B 0,C 180,E1 18903.8,E2 18903.8} C_VEL
LIN {X 0,Y 392.121,Z 791.654,A -85,B 0,C 180,E1 18901.169,E2 18901.169} C_VEL
LIN {X 0,Y 392.098,Z 791.238,A -85,B 0,C 180,E1 18898.539,E2 18898.539} C_VEL
LIN {X 0,Y 392.134,Z 789.144,A -85,B 0,C 180,E1 18895.906,E2 18895.906} C_VEL
LIN {X 0,Y 392.276,Z 785.324,A -85,B 0,C 180,E1 18893.267,E2 18893.267} C_VEL
LIN {X 0,Y 392.586,Z 779.679,A -85,B 0,C 180,E1 18890.619,E2 18890.619} C_VEL
LIN {X 0,Y 393.102,Z 772.527,A -85,B 0,C 180,E1 18888.11,E2 18888.11} C_VEL
LIN {X 0,Y 393.92,Z 763.387,A -85,B 0,C 180,E1 18885.596,E2 18885.596} C_VEL
LIN {X 0,Y 395.012,Z 752.673,A -85,B 0,C 180,E1 18883.228,E2 18883.228} C_VEL
LIN {X 0,Y 396.361,Z 740.413,A -85,B 0,C 180,E1 18881.009,E2 18881.009} C_VEL
LIN {X 0,Y 397.925,Z 726.489,A -85,B 0,C 180,E1 18878.942,E2 18878.942} C_VEL
LIN {X 0,Y 399.596,Z 711.46,A -85,B 0,C 180,E1 18877.102,E2 18877.102} C_VEL
LIN {X 0,Y 401.28,Z 695.458,A -85,B 0,C 180,E1 18875.489,E2 18875.489} C_VEL
LIN {X 0,Y 402.996,Z 677.67,A -85,B 0,C 180,E1 18874.035,E2 18874.035} C_VEL
LIN {X 0,Y 404.546,Z 659.247,A -85,B 0,C 180,E1 18872.844,E2 18872.844} C_VEL
LIN {X 0,Y 405.877,Z 639.977,A -85,B 0,C 180,E1 18871.896,E2 18871.896} C_VEL
LIN {X 0,Y 406.872,Z 620.315,A -85,B 0,C 180,E1 18871.216,E2 18871.216} C_VEL
LIN {X 0,Y 413.234,Z 436.014,A -85,B 0,C 180,E1 18867.214,E2 18867.214} C_VEL
LIN {X 0,Y 410.91,Z 423.442,A -85,B 0,C 180,E1 18866.719,E2 18866.719} C_VEL
LIN {X 0,Y 404.687,Z 410.112,A -85,B 0,C 180,E1 18865.862,E2 18865.862} C_VEL
LIN {X 0,Y 397.437,Z 388.951,A -85,B 0,C 180,E1 18862.858,E2 18862.858} C_VEL
LIN {X 0,Y 393.503,Z 377.784,A -85,B 0,C 180,E1 18861.219,E2 18861.219} C_VEL
LIN {X 0,Y 393.497,Z 377.782,A -85,B 0,C 180,E1 18857.467,E2 18857.467} C_VEL
LIN {X 0,Y 393.497,Z 377.781,A -85,B 0,C 180,E1 18853.52,E2 18853.52} C_VEL
LIN {X 0,Y 393.499,Z 377.781,A -85,B 0,C 180,E1 18849.627,E2 18849.627} C_VEL
LIN {X 0,Y 393.507,Z 377.782,A -85,B 0,C 180,E1 18845.761,E2 18845.761} C_VEL
LIN {X 0,Y 393.518,Z 377.78,A -85,B 0,C 180,E1 18841.904,E2 18841.904} C_VEL
LIN {X 0,Y 393.533,Z 377.78,A -85,B 0,C 180,E1 18838.037,E2 18838.037} C_VEL
LIN {X 0,Y 393.54,Z 377.776,A -85,B 0,C 180,E1 18834.145,E2 18834.145} C_VEL
LIN {X 0,Y 393.542,Z 377.776,A -85,B 0,C 180,E1 18830.214,E2 18830.214} C_VEL
LIN {X 0,Y 393.542,Z 377.776,A -85,B 0,C 180,E1 18826.183,E2 18826.183} C_VEL
LIN {X 0,Y 393.528,Z 377.775,A -85,B 0,C 180,E1 18822.323,E2 18822.323} C_VEL
LIN {X 0,Y 393.515,Z 377.776,A -85,B 0,C 180,E1 18819.648,E2 18819.648} C_VEL
LIN {X 0,Y 392.466,Z 377.906,A -85,B 0,C 180,E1 18818.527,E2 18818.527} C_VEL
LIN {X 0,Y 385.969,Z 378.717,A -85,B 0,C 180,E1 18815.281,E2 18815.281} C_VEL
LIN {X 0,Y 385.568,Z 378.766,A -85,B 0,C 180,E1 18814.536,E2 18814.536} C_VEL
LIN {X 0,Y 385.561,Z 378.768,A -85,B 0,C 180,E1 18810.594,E2 18810.594} C_VEL
LIN {X 0,Y 385.556,Z 378.764,A -85,B 0,C 180,E1 18806.729,E2 18806.729} C_VEL
LIN {X 0,Y 385.553,Z 378.764,A -85,B 0,C 180,E1 18802.849,E2 18802.849} C_VEL
LIN {X 0,Y 385.555,Z 378.768,A -85,B 0,C 180,E1 18798.785,E2 18798.785} C_VEL
LIN {X 0,Y 385.554,Z 378.77,A -85,B 0,C 180,E1 18794.734,E2 18794.734} C_VEL
LIN {X 0,Y 385.556,Z 378.77,A -85,B 0,C 180,E1 18790.728,E2 18790.728} C_VEL
LIN {X 0,Y 385.556,Z 378.768,A -85,B 0,C 180,E1 18786.64,E2 18786.64} C_VEL
LIN {X 0,Y 385.556,Z 378.768,A -85,B 0,C 180,E1 18782.676,E2 18782.676} C_VEL
LIN {X 0,Y 385.556,Z 378.77,A -85,B 0,C 180,E1 18778.561,E2 18778.561} C_VEL
LIN {X 0,Y 385.554,Z 378.774,A -85,B 0,C 180,E1 18774.486,E2 18774.486} C_VEL
LIN {X 0,Y 385.555,Z 378.772,A -85,B 0,C 180,E1 18770.553,E2 18770.553} C_VEL
LIN {X 0,Y 385.553,Z 378.771,A -85,B 0,C 180,E1 18766.563,E2 18766.563} C_VEL
LIN {X 0,Y 385.555,Z 378.772,A -85,B 0,C 180,E1 18762.566,E2 18762.566} C_VEL
LIN {X 0,Y 385.555,Z 378.773,A -85,B 0,C 180,E1 18758.681,E2 18758.681} C_VEL
LIN {X 0,Y 385.586,Z 378.834,A -85,B 0,C 180,E1 18757.73,E2 18757.73} C_VEL
LIN {X 0,Y 390.944,Z 397.81,A -85,B 0,C 180,E1 18754.039,E2 18754.039} C_VEL
LIN {X 0,Y 395.546,Z 415.769,A -85,B 0,C 180,E1 18750.744,E2 18750.744} C_VEL
LIN {X 0,Y 393.041,Z 442.53,A -85,B 0,C 180,E1 18746.68,E2 18746.68} C_VEL
LIN {X 0,Y 390.665,Z 470.986,A -85,B 0,C 180,E1 18742.417,E2 18742.417} C_VEL
LIN {X 0,Y 390.149,Z 478.641,A -85,B 0,C 180,E1 18741.319,E2 18741.319} C_VEL
LIN {X 0,Y 393.716,Z 506.183,A -85,B 0,C 180,E1 18740.409,E2 18740.409} C_VEL
LIN {X 0,Y 390.756,Z 604.557,A -85,B 0,C 180,E1 18737.978,E2 18737.978} C_VEL
LIN {X 0,Y 390.263,Z 620.444,A -85,B 0,C 180,E1 18737.328,E2 18737.328} C_VEL
LIN {X 0,Y 389.591,Z 636.313,A -85,B 0,C 180,E1 18736.398,E2 18736.398} C_VEL
LIN {X 0,Y 388.727,Z 652.052,A -85,B 0,C 180,E1 18735.153,E2 18735.153} C_VEL
LIN {X 0,Y 387.921,Z 665.97,A -85,B 0,C 180,E1 18733.717,E2 18733.717} C_VEL
LIN {X 0,Y 387.19,Z 677.995,A -85,B 0,C 180,E1 18732.15,E2 18732.15} C_VEL
LIN {X 0,Y 386.561,Z 688.572,A -85,B 0,C 180,E1 18730.432,E2 18730.432} C_VEL
LIN {X 0,Y 386.043,Z 697.978,A -85,B 0,C 180,E1 18728.49,E2 18728.49} C_VEL
LIN {X 0,Y 385.708,Z 705.211,A -85,B 0,C 180,E1 18726.55,E2 18726.55} C_VEL
LIN {X 0,Y 385.521,Z 711.055,A -85,B 0,C 180,E1 18724.463,E2 18724.463} C_VEL
LIN {X 0,Y 385.488,Z 715.204,A -85,B 0,C 180,E1 18722.23,E2 18722.23} C_VEL
LIN {X 0,Y 385.578,Z 717.306,A -85,B 0,C 180,E1 18720.149,E2 18720.149} C_VEL
LIN {X 0,Y 385.831,Z 717.72,A -85,B 0,C 180,E1 18717.921,E2 18717.921} C_VEL
LIN {X 0,Y 386.184,Z 716.336,A -85,B 0,C 180,E1 18715.843,E2 18715.843} C_VEL
LIN {X 0,Y 386.766,Z 712.964,A -85,B 0,C 180,E1 18713.618,E2 18713.618} C_VEL
LIN {X 0,Y 387.509,Z 707.871,A -85,B 0,C 180,E1 18711.543,E2 18711.543} C_VEL
LIN {X 0,Y 388.404,Z 701.358,A -85,B 0,C 180,E1 18709.619,E2 18709.619} C_VEL
LIN {X 0,Y 389.514,Z 692.685,A -85,B 0,C 180,E1 18707.699,E2 18707.699} C_VEL
LIN {X 0,Y 390.768,Z 682.492,A -85,B 0,C 180,E1 18705.932,E2 18705.932} C_VEL
LIN {X 0,Y 392.099,Z 670.744,A -85,B 0,C 180,E1 18704.318,E2 18704.318} C_VEL
LIN {X 0,Y 393.508,Z 656.801,A -85,B 0,C 180,E1 18702.82,E2 18702.82} C_VEL
LIN {X 0,Y 394.913,Z 641.649,A -85,B 0,C 180,E1 18701.55,E2 18701.55} C_VEL
LIN {X 0,Y 396.128,Z 625.739,A -85,B 0,C 180,E1 18700.538,E2 18700.538} C_VEL
LIN {X 0,Y 397.164,Z 608.998,A -85,B 0,C 180,E1 18699.767,E2 18699.767} C_VEL
LIN {X 0,Y 404.457,Z 520.984,A -85,B 0,C 180,E1 18696.744,E2 18696.744} C_VEL
LIN {X 0,Y 405.247,Z 510.722,A -85,B 0,C 180,E1 18696.372,E2 18696.372} C_VEL
LIN {X 0,Y 402.673,Z 491.838,A -85,B 0,C 180,E1 18695.103,E2 18695.103} C_VEL
LIN {X 0,Y 400.237,Z 478.046,A -85,B 0,C 180,E1 18693.996,E2 18693.996} C_VEL
LIN {X 0,Y 405.389,Z 454.396,A -85,B 0,C 180,E1 18689.792,E2 18689.792} C_VEL
LIN {X 0,Y 409.665,Z 439.378,A -85,B 0,C 180,E1 18686.942,E2 18686.942} C_VEL
LIN {X 0,Y 409.043,Z 433.344,A -85,B 0,C 180,E1 18684.94,E2 18684.94} C_VEL
LIN {X 0,Y 408.303,Z 428.064,A -85,B 0,C 180,E1 18682.605,E2 18682.605} C_VEL
LIN {X 0,Y 407.897,Z 424.556,A -85,B 0,C 180,E1 18680.225,E2 18680.225} C_VEL
LIN {X 0,Y 408.061,Z 422.826,A -85,B 0,C 180,E1 18677.447,E2 18677.447} C_VEL
LIN {X 0,Y 408.371,Z 423.266,A -85,B 0,C 180,E1 18675.945,E2 18675.945} C_VEL
LIN {X 0,Y 409.385,Z 426.126,A -85,B 0,C 180,E1 18673.296,E2 18673.296} C_VEL
LIN {X 0,Y 410.721,Z 430.784,A -85,B 0,C 180,E1 18671.094,E2 18671.094} C_VEL
LIN {X 0,Y 412.186,Z 436.392,A -85,B 0,C 180,E1 18669.204,E2 18669.204} C_VEL
LIN {X 0,Y 412.898,Z 440.049,A -85,B 0,C 180,E1 18668.231,E2 18668.231} C_VEL
LIN {X 0,Y 406.714,Z 462.307,A -85,B 0,C 180,E1 18665.291,E2 18665.291} C_VEL
LIN {X 0,Y 405.19,Z 469.829,A -85,B 0,C 180,E1 18664.383,E2 18664.383} C_VEL
LIN {X 0,Y 406.358,Z 482.056,A -85,B 0,C 180,E1 18663.781,E2 18663.781} C_VEL
LIN {X 0,Y 406.816,Z 493.535,A -85,B 0,C 180,E1 18663.32,E2 18663.32} C_VEL
LIN {X 0,Y 401.948,Z 584.22,A -85,B 0,C 180,E1 18661.034,E2 18661.034} C_VEL
LIN {X 0,Y 398.916,Z 660.764,A -85,B 0,C 180,E1 18659.244,E2 18659.244} C_VEL
LIN {X 0,Y 396.973,Z 688.616,A -85,B 0,C 180,E1 18658.212,E2 18658.212} C_VEL
LIN {X 0,Y 395.413,Z 707.484,A -85,B 0,C 180,E1 18657.238,E2 18657.238} C_VEL
LIN {X 0,Y 393.744,Z 724.988,A -85,B 0,C 180,E1 18656.06,E2 18656.06} C_VEL
LIN {X 0,Y 391.923,Z 742.57,A -85,B 0,C 180,E1 18654.572,E2 18654.572} C_VEL
LIN {X 0,Y 390.115,Z 758.937,A -85,B 0,C 180,E1 18652.848,E2 18652.848} C_VEL
LIN {X 0,Y 388.478,Z 773.653,A -85,B 0,C 180,E1 18650.963,E2 18650.963} C_VEL
LIN {X 0,Y 387.022,Z 787.329,A -85,B 0,C 180,E1 18648.841,E2 18648.841} C_VEL
LIN {X 0,Y 385.832,Z 799.429,A -85,B 0,C 180,E1 18646.562,E2 18646.562} C_VEL
LIN {X 0,Y 384.989,Z 809.98,A -85,B 0,C 180,E1 18644.13,E2 18644.13} C_VEL
LIN {X 0,Y 384.463,Z 818.446,A -85,B 0,C 180,E1 18641.704,E2 18641.704} C_VEL
LIN {X 0,Y 384.217,Z 825.467,A -85,B 0,C 180,E1 18639.134,E2 18639.134} C_VEL
LIN {X 0,Y 384.171,Z 830.636,A -85,B 0,C 180,E1 18636.576,E2 18636.576} C_VEL
LIN {X 0,Y 384.213,Z 834.077,A -85,B 0,C 180,E1 18634.029,E2 18634.029} C_VEL
LIN {X 0,Y 384.273,Z 835.872,A -85,B 0,C 180,E1 18631.491,E2 18631.491} C_VEL
LIN {X 0,Y 384.282,Z 836.055,A -85,B 0,C 180,E1 18628.956,E2 18628.956} C_VEL
LIN {X 0,Y 384.216,Z 834.499,A -85,B 0,C 180,E1 18626.27,E2 18626.27} C_VEL
LIN {X 0,Y 384.162,Z 831.125,A -85,B 0,C 180,E1 18623.574,E2 18623.574} C_VEL
LIN {X 0,Y 384.201,Z 826.212,A -85,B 0,C 180,E1 18621.017,E2 18621.017} C_VEL
LIN {X 0,Y 384.447,Z 819.504,A -85,B 0,C 180,E1 18618.448,E2 18618.448} C_VEL
LIN {X 0,Y 385.012,Z 810.852,A -85,B 0,C 180,E1 18615.87,E2 18615.87} C_VEL
LIN {X 0,Y 385.899,Z 800.701,A -85,B 0,C 180,E1 18613.441,E2 18613.441} C_VEL
LIN {X 0,Y 387.14,Z 789.128,A -85,B 0,C 180,E1 18611.165,E2 18611.165} C_VEL
LIN {X 0,Y 388.687,Z 776.064,A -85,B 0,C 180,E1 18609.032,E2 18609.032} C_VEL
LIN {X 0,Y 390.565,Z 761.251,A -85,B 0,C 180,E1 18607.02,E2 18607.02} C_VEL
LIN {X 0,Y 392.614,Z 745.363,A -85,B 0,C 180,E1 18605.233,E2 18605.233} C_VEL
LIN {X 0,Y 394.839,Z 727.738,A -85,B 0,C 180,E1 18603.613,E2 18603.613} C_VEL
LIN {X 0,Y 397.1,Z 709.139,A -85,B 0,C 180,E1 18602.237,E2 18602.237} C_VEL
LIN {X 0,Y 399.311,Z 689.572,A -85,B 0,C 180,E1 18601.101,E2 18601.101} C_VEL
LIN {X 0,Y 401.395,Z 668.823,A -85,B 0,C 180,E1 18600.202,E2 18600.202} C_VEL
LIN {X 0,Y 403.143,Z 644.035,A -85,B 0,C 180,E1 18599.461,E2 18599.461} C_VEL
LIN {X 0,Y 408.362,Z 569.185,A -85,B 0,C 180,E1 18597.378,E2 18597.378} C_VEL
LIN {X 0,Y 415.324,Z 492.716,A -85,B 0,C 180,E1 18595.09,E2 18595.09} C_VEL
LIN {X 0,Y 415.112,Z 464.142,A -85,B 0,C 180,E1 18593.55,E2 18593.55} C_VEL
LIN {X 0,Y 414.962,Z 438.361,A -85,B 0,C 180,E1 18591.892,E2 18591.892} C_VEL
LIN {X 0,Y 414.88,Z 435.624,A -85,B 0,C 180,E1 18591.62,E2 18591.62} C_VEL
LIN {X 0,Y 412.882,Z 423.847,A -85,B 0,C 180,E1 18589.633,E2 18589.633} C_VEL
LIN {X 0,Y 412.49,Z 416.56,A -85,B 0,C 180,E1 18588.195,E2 18588.195} C_VEL
LIN {X 0,Y 412.367,Z 415.136,A -85,B 0,C 180,E1 18587.806,E2 18587.806} C_VEL
LIN {X 0,Y 410.985,Z 413.487,A -85,B 0,C 180,E1 18585.864,E2 18585.864} C_VEL
LIN {X 0,Y 410.5,Z 413.981,A -85,B 0,C 180,E1 18583.865,E2 18583.865} C_VEL
LIN {X 0,Y 411.07,Z 415.516,A -85,B 0,C 180,E1 18582.169,E2 18582.169} C_VEL
LIN {X 0,Y 412.04,Z 419.26,A -85,B 0,C 180,E1 18580.363,E2 18580.363} C_VEL
LIN {X 0,Y 413.704,Z 424.854,A -85,B 0,C 180,E1 18578.458,E2 18578.458} C_VEL
LIN {X 0,Y 417.361,Z 432.853,A -85,B 0,C 180,E1 18576.814,E2 18576.814} C_VEL
LIN {X 0,Y 420.241,Z 440.193,A -85,B 0,C 180,E1 18575.694,E2 18575.694} C_VEL
LIN {X 0,Y 420.247,Z 443.938,A -85,B 0,C 180,E1 18575.482,E2 18575.482} C_VEL
LIN {X 0,Y 411.25,Z 529.063,A -85,B 0,C 180,E1 18572.93,E2 18572.93} C_VEL
LIN {X 0,Y 405.438,Z 602.661,A -85,B 0,C 180,E1 18570.84,E2 18570.84} C_VEL
LIN {X 0,Y 403.587,Z 631.651,A -85,B 0,C 180,E1 18569.983,E2 18569.983} C_VEL
LIN {X 0,Y 402,Z 651.202,A -85,B 0,C 180,E1 18569.135,E2 18569.135} C_VEL
LIN {X 0,Y 400.108,Z 670.392,A -85,B 0,C 180,E1 18568.022,E2 18568.022} C_VEL
LIN {X 0,Y 397.992,Z 688.753,A -85,B 0,C 180,E1 18566.655,E2 18566.655} C_VEL
LIN {X 0,Y 395.827,Z 705.351,A -85,B 0,C 180,E1 18565.11,E2 18565.11} C_VEL
LIN {X 0,Y 393.649,Z 720.887,A -85,B 0,C 180,E1 18563.343,E2 18563.343} C_VEL
LIN {X 0,Y 391.515,Z 735.366,A -85,B 0,C 180,E1 18561.341,E2 18561.341} C_VEL
LIN {X 0,Y 389.59,Z 748.241,A -85,B 0,C 180,E1 18559.178,E2 18559.178} C_VEL
LIN {X 0,Y 387.879,Z 759.91,A -85,B 0,C 180,E1 18556.781,E2 18556.781} C_VEL
LIN {X 0,Y 386.558,Z 769.343,A -85,B 0,C 180,E1 18554.377,E2 18554.377} C_VEL
LIN {X 0,Y 385.54,Z 777.31,A -85,B 0,C 180,E1 18551.822,E2 18551.822} C_VEL
LIN {X 0,Y 384.842,Z 783.678,A -85,B 0,C 180,E1 18549.147,E2 18549.147} C_VEL
LIN {X 0,Y 384.428,Z 788.279,A -85,B 0,C 180,E1 18546.421,E2 18546.421} C_VEL
LIN {X 0,Y 384.221,Z 791.071,A -85,B 0,C 180,E1 18543.73,E2 18543.73} C_VEL
LIN {X 0,Y 384.136,Z 792.171,A -85,B 0,C 180,E1 18541.044,E2 18541.044} C_VEL
LIN {X 0,Y 384.111,Z 791.578,A -85,B 0,C 180,E1 18538.334,E2 18538.334} C_VEL
LIN {X 0,Y 384.154,Z 789.329,A -85,B 0,C 180,E1 18535.671,E2 18535.671} C_VEL
LIN {X 0,Y 384.317,Z 785.328,A -85,B 0,C 180,E1 18532.976,E2 18532.976} C_VEL
LIN {X 0,Y 384.663,Z 779.485,A -85,B 0,C 180,E1 18530.273,E2 18530.273} C_VEL
LIN {X 0,Y 385.237,Z 772.115,A -85,B 0,C 180,E1 18527.712,E2 18527.712} C_VEL
LIN {X 0,Y 386.062,Z 763.322,A -85,B 0,C 180,E1 18525.297,E2 18525.297} C_VEL
LIN {X 0,Y 387.221,Z 752.466,A -85,B 0,C 180,E1 18522.88,E2 18522.88} C_VEL
LIN {X 0,Y 388.645,Z 739.991,A -85,B 0,C 180,E1 18520.617,E2 18520.617} C_VEL
LIN {X 0,Y 390.238,Z 726.36,A -85,B 0,C 180,E1 18518.579,E2 18518.579} C_VEL
LIN {X 0,Y 391.983,Z 711.242,A -85,B 0,C 180,E1 18516.711,E2 18516.711} C_VEL
LIN {X 0,Y 393.807,Z 694.503,A -85,B 0,C 180,E1 18515.014,E2 18515.014} C_VEL
LIN {X 0,Y 395.546,Z 677.049,A -85,B 0,C 180,E1 18513.583,E2 18513.583} C_VEL
LIN {X 0,Y 397.118,Z 658.882,A -85,B 0,C 180,E1 18512.401,E2 18512.401} C_VEL
LIN {X 0,Y 398.474,Z 639.708,A -85,B 0,C 180,E1 18511.453,E2 18511.453} C_VEL
LIN {X 0,Y 399.504,Z 620.053,A -85,B 0,C 180,E1 18510.768,E2 18510.768} C_VEL
LIN {X 0,Y 406.178,Z 437.171,A -85,B 0,C 180,E1 18506.692,E2 18506.692} C_VEL
LIN {X 0,Y 404.165,Z 426.475,A -85,B 0,C 180,E1 18506.257,E2 18506.257} C_VEL
LIN {X 0,Y 396.668,Z 410.496,A -85,B 0,C 180,E1 18505.196,E2 18505.196} C_VEL
LIN {X 0,Y 389.324,Z 389.297,A -85,B 0,C 180,E1 18502.135,E2 18502.135} C_VEL
LIN {X 0,Y 385.61,Z 378.761,A -85,B 0,C 180,E1 18500.56,E2 18500.56} C_VEL
LIN {X 0,Y 385.6,Z 378.769,A -85,B 0,C 180,E1 18496.556,E2 18496.556} C_VEL
LIN {X 0,Y 385.597,Z 378.767,A -85,B 0,C 180,E1 18492.573,E2 18492.573} C_VEL
LIN {X 0,Y 385.588,Z 378.769,A -85,B 0,C 180,E1 18488.677,E2 18488.677} C_VEL
LIN {X 0,Y 385.58,Z 378.771,A -85,B 0,C 180,E1 18484.712,E2 18484.712} C_VEL
LIN {X 0,Y 385.578,Z 378.769,A -85,B 0,C 180,E1 18480.721,E2 18480.721} C_VEL
